LIN {X 0,Y 216.17,Z 835.857,A -85,B 0,C 180,E1 9801.223,E2 9801.223} C_VEL
LIN {X 0,Y 213.563,Z 840.911,A -85,B 0,C 180,E1 9796.189,E2 9796.189} C_VEL
LIN {X 0,Y 211.955,Z 844.646,A -85,B 0,C 180,E1 9790.637,E2 9790.637} C_VEL
LIN {X 0,Y 211.434,Z 846.63,A -85,B 0,C 180,E1 9785.221,E2 9785.221} C_VEL
LIN {X 0,Y 211.788,Z 847.099,A -85,B 0,C 180,E1 9779.975,E2 9779.975} C_VEL
LIN {X 0,Y 213.212,Z 845.891,A -85,B 0,C 180,E1 9774.219,E2 9774.219} C_VEL
LIN {X 0,Y 215.988,Z 842.864,A -85,B 0,C 180,E1 9768.553,E2 9768.553} C_VEL
LIN {X 0,Y 219.977,Z 838.26,A -85,B 0,C 180,E1 9763.339,E2 9763.339} C_VEL
LIN {X 0,Y 225.319,Z 832.008,A -85,B 0,C 180,E1 9758.406,E2 9758.406} C_VEL
LIN {X 0,Y 231.998,Z 823.945,A -85,B 0,C 180,E1 9753.723,E2 9753.723} C_VEL
LIN {X 0,Y 239.833,Z 814.067,A -85,B 0,C 180,E1 9749.394,E2 9749.394} C_VEL
LIN {X 0,Y 248.295,Z 802.757,A -85,B 0,C 180,E1 9745.582,E2 9745.582} C_VEL
LIN {X 0,Y 257.088,Z 790.107,A -85,B 0,C 180,E1 9742.245,E2 9742.245} C_VEL
LIN {X 0,Y 266.114,Z 775.981,A -85,B 0,C 180,E1 9739.307,E2 9739.307} C_VEL
LIN {X 0,Y 275.138,Z 760.195,A -85,B 0,C 180,E1 9736.725,E2 9736.725} C_VEL
LIN {X 0,Y 283.583,Z 743.647,A -85,B 0,C 180,E1 9734.582,E2 9734.582} C_VEL
LIN {X 0,Y 291.207,Z 726.587,A -85,B 0,C 180,E1 9732.821,E2 9732.821} C_VEL
LIN {X 0,Y 298.253,Z 708.268,A -85,B 0,C 180,E1 9731.326,E2 9731.326} C_VEL
LIN {X 0,Y 304.418,Z 689.211,A -85,B 0,C 180,E1 9730.108,E2 9730.108} C_VEL
LIN {X 0,Y 309.578,Z 669.056,A -85,B 0,C 180,E1 9729.137,E2 9729.137} C_VEL
LIN {X 0,Y 313.491,Z 648.587,A -85,B 0,C 180,E1 9728.428,E2 9728.428} C_VEL
LIN {X 0,Y 315.036,Z 637.769,A -85,B 0,C 180,E1 9728.146,E2 9728.146} C_VEL
LIN {X 0,Y 315.658,Z 630.27,A -85,B 0,C 180,E1 9727.794,E2 9727.794} C_VEL
LIN {X 0,Y 316.044,Z 610.74,A -85,B 0,C 180,E1 9726.277,E2 9726.277} C_VEL
LIN {X 0,Y 316.562,Z 604.27,A -85,B 0,C 180,E1 9726.008,E2 9726.008} C_VEL
LIN {X 0,Y 330.668,Z 479.091,A -85,B 0,C 180,E1 9723.364,E2 9723.364} C_VEL
LIN {X 0,Y 333.385,Z 441.647,A -85,B 0,C 180,E1 9721.202,E2 9721.202} C_VEL
LIN {X 0,Y 332.154,Z 436.517,A -85,B 0,C 180,E1 9718.878,E2 9718.878} C_VEL
LIN {X 0,Y 331.429,Z 432.32,A -85,B 0,C 180,E1 9716.107,E2 9716.107} C_VEL
LIN {X 0,Y 331.783,Z 429.625,A -85,B 0,C 180,E1 9712.38,E2 9712.38} C_VEL
LIN {X 0,Y 332.681,Z 430.118,A -85,B 0,C 180,E1 9710.135,E2 9710.135} C_VEL
LIN {X 0,Y 334.995,Z 433.817,A -85,B 0,C 180,E1 9706.801,E2 9706.801} C_VEL
LIN {X 0,Y 336.697,Z 436.983,A -85,B 0,C 180,E1 9705.066,E2 9705.066} C_VEL
LIN {X 0,Y 321.679,Z 592.371,A -85,B 0,C 180,E1 9701.883,E2 9701.883} C_VEL
LIN {X 0,Y 316.022,Z 652.978,A -85,B 0,C 180,E1 9700.612,E2 9700.612} C_VEL
LIN {X 0,Y 312.317,Z 675.121,A -85,B 0,C 180,E1 9699.999,E2 9699.999} C_VEL
LIN {X 0,Y 307.316,Z 696.218,A -85,B 0,C 180,E1 9699.228,E2 9699.228} C_VEL
LIN {X 0,Y 301.4,Z 716.25,A -85,B 0,C 180,E1 9698.252,E2 9698.252} C_VEL
LIN {X 0,Y 294.376,Z 735.972,A -85,B 0,C 180,E1 9697.008,E2 9697.008} C_VEL
LIN {X 0,Y 286.184,Z 755.614,A -85,B 0,C 180,E1 9695.432,E2 9695.432} C_VEL
LIN {X 0,Y 277.441,Z 774.165,A -85,B 0,C 180,E1 9693.569,E2 9693.569} C_VEL
LIN {X 0,Y 268.335,Z 791.382,A -85,B 0,C 180,E1 9691.402,E2 9691.402} C_VEL
LIN {X 0,Y 257.843,Z 809.537,A -85,B 0,C 180,E1 9688.546,E2 9688.546} C_VEL
LIN {X 0,Y 247.851,Z 825.668,A -85,B 0,C 180,E1 9685.377,E2 9685.377} C_VEL
LIN {X 0,Y 237.561,Z 841.407,A -85,B 0,C 180,E1 9681.47,E2 9681.47} C_VEL
LIN {X 0,Y 228.085,Z 855.483,A -85,B 0,C 180,E1 9677.057,E2 9677.057} C_VEL
LIN {X 0,Y 219.562,Z 868.331,A -85,B 0,C 180,E1 9672.018,E2 9672.018} C_VEL
LIN {X 0,Y 212.413,Z 879.754,A -85,B 0,C 180,E1 9666.373,E2 9666.373} C_VEL
LIN {X 0,Y 207.135,Z 889.148,A -85,B 0,C 180,E1 9660.45,E2 9660.45} C_VEL
LIN {X 0,Y 203.464,Z 897.482,A -85,B 0,C 180,E1 9653.76,E2 9653.76} C_VEL
LIN {X 0,Y 201.898,Z 903.094,A -85,B 0,C 180,E1 9647.878,E2 9647.878} C_VEL
LIN {X 0,Y 201.535,Z 907.332,A -85,B 0,C 180,E1 9641.733,E2 9641.733} C_VEL
LIN {X 0,Y 201.829,Z 909.538,A -85,B 0,C 180,E1 9636.825,E2 9636.825} C_VEL
LIN {X 0,Y 202.15,Z 910.582,A -85,B 0,C 180,E1 9632.265,E2 9632.265} C_VEL
LIN {X 0,Y 202.167,Z 910.586,A -85,B 0,C 180,E1 9628.013,E2 9628.013} C_VEL
LIN {X 0,Y 201.84,Z 909.458,A -85,B 0,C 180,E1 9623.169,E2 9623.169} C_VEL
LIN {X 0,Y 201.572,Z 906.678,A -85,B 0,C 180,E1 9617.682,E2 9617.682} C_VEL
LIN {X 0,Y 201.959,Z 902.561,A -85,B 0,C 180,E1 9612.122,E2 9612.122} C_VEL
LIN {X 0,Y 203.657,Z 896.224,A -85,B 0,C 180,E1 9605.948,E2 9605.948} C_VEL
LIN {X 0,Y 206.793,Z 888.559,A -85,B 0,C 180,E1 9600.128,E2 9600.128} C_VEL
LIN {X 0,Y 211.703,Z 878.744,A -85,B 0,C 180,E1 9594.326,E2 9594.326} C_VEL
LIN {X 0,Y 218.021,Z 867.475,A -85,B 0,C 180,E1 9589.016,E2 9589.016} C_VEL
LIN {X 0,Y 225.224,Z 855.274,A -85,B 0,C 180,E1 9584.375,E2 9584.375} C_VEL
LIN {X 0,Y 233.702,Z 840.845,A -85,B 0,C 180,E1 9580.016,E2 9580.016} C_VEL
LIN {X 0,Y 242.489,Z 825.468,A -85,B 0,C 180,E1 9576.279,E2 9576.279} C_VEL
LIN {X 0,Y 251.282,Z 809.376,A -85,B 0,C 180,E1 9573.117,E2 9573.117} C_VEL
LIN {X 0,Y 260.122,Z 791.762,A -85,B 0,C 180,E1 9570.349,E2 9570.349} C_VEL
LIN {X 0,Y 268.829,Z 772.701,A -85,B 0,C 180,E1 9567.946,E2 9567.946} C_VEL
LIN {X 0,Y 276.623,Z 753.661,A -85,B 0,C 180,E1 9566.014,E2 9566.014} C_VEL
LIN {X 0,Y 283.429,Z 734.543,A -85,B 0,C 180,E1 9564.47,E2 9564.47} C_VEL
LIN {X 0,Y 289.725,Z 713.651,A -85,B 0,C 180,E1 9563.138,E2 9563.138} C_VEL
LIN {X 0,Y 295.057,Z 692.142,A -85,B 0,C 180,E1 9562.083,E2 9562.083} C_VEL
LIN {X 0,Y 299.172,Z 670.359,A -85,B 0,C 180,E1 9561.305,E2 9561.305} C_VEL
LIN {X 0,Y 301.898,Z 648.014,A -85,B 0,C 180,E1 9560.706,E2 9560.706} C_VEL
LIN {X 0,Y 316.697,Z 449.988,A -85,B 0,C 180,E1 9556.577,E2 9556.577} C_VEL
LIN {X 0,Y 318.4,Z 427.647,A -85,B 0,C 180,E1 9556.089,E2 9556.089} C_VEL
LIN {X 0,Y 309.751,Z 414.232,A -85,B 0,C 180,E1 9552.443,E2 9552.443} C_VEL
LIN {X 0,Y 301.912,Z 402.88,A -85,B 0,C 180,E1 9548.667,E2 9548.667} C_VEL
LIN {X 0,Y 294.659,Z 393.174,A -85,B 0,C 180,E1 9544.574,E2 9544.574} C_VEL
LIN {X 0,Y 289.984,Z 387.27,A -85,B 0,C 180,E1 9541.492,E2 9541.492} C_VEL
LIN {X 0,Y 287.159,Z 383.801,A -85,B 0,C 180,E1 9539.402,E2 9539.402} C_VEL
LIN {X 0,Y 283.546,Z 379.395,A -85,B 0,C 180,E1 9536.337,E2 9536.337} C_VEL
LIN {X 0,Y 279.243,Z 374.32,A -85,B 0,C 180,E1 9531.766,E2 9531.766} C_VEL
LIN {X 0,Y 274.47,Z 369.423,A -85,B 0,C 180,E1 9523.057,E2 9523.057} C_VEL
LIN {X 0,Y 273.587,Z 369.085,A -85,B 0,C 180,E1 9519.238,E2 9519.238} C_VEL
LIN {X 0,Y 273.555,Z 370.592,A -85,B 0,C 180,E1 9514.915,E2 9514.915} C_VEL
LIN {X 0,Y 275.286,Z 373.534,A -85,B 0,C 180,E1 9509.075,E2 9509.075} C_VEL
LIN {X 0,Y 278.207,Z 378.589,A -85,B 0,C 180,E1 9504.141,E2 9504.141} C_VEL
LIN {X 0,Y 281.069,Z 383.491,A -85,B 0,C 180,E1 9500.642,E2 9500.642} C_VEL
LIN {X 0,Y 284.697,Z 389.345,A -85,B 0,C 180,E1 9497.191,E2 9497.191} C_VEL
LIN {X 0,Y 290.304,Z 398.667,A -85,B 0,C 180,E1 9492.892,E2 9492.892} C_VEL
LIN {X 0,Y 296.513,Z 409.789,A -85,B 0,C 180,E1 9488.915,E2 9488.915} C_VEL
LIN {X 0,Y 301.972,Z 420.129,A -85,B 0,C 180,E1 9485.903,E2 9485.903} C_VEL
LIN {X 0,Y 303.039,Z 422.43,A -85,B 0,C 180,E1 9485.339,E2 9485.339} C_VEL
LIN {X 0,Y 302.745,Z 475.251,A -85,B 0,C 180,E1 9482.474,E2 9482.474} C_VEL
LIN {X 0,Y 287.453,Z 637.405,A -85,B 0,C 180,E1 9478.809,E2 9478.809} C_VEL
LIN {X 0,Y 284.269,Z 658.885,A -85,B 0,C 180,E1 9478.1,E2 9478.1} C_VEL
LIN {X 0,Y 280.102,Z 679.277,A -85,B 0,C 180,E1 9477.133,E2 9477.133} C_VEL
LIN {X 0,Y 274.985,Z 699.045,A -85,B 0,C 180,E1 9475.872,E2 9475.872} C_VEL
LIN {X 0,Y 268.872,Z 718.482,A -85,B 0,C 180,E1 9474.265,E2 9474.265} C_VEL
LIN {X 0,Y 262.041,Z 736.952,A -85,B 0,C 180,E1 9472.315,E2 9472.315} C_VEL
LIN {X 0,Y 255.013,Z 753.63,A -85,B 0,C 180,E1 9470.102,E2 9470.102} C_VEL
LIN {X 0,Y 247.357,Z 769.856,A -85,B 0,C 180,E1 9467.407,E2 9467.407} C_VEL
LIN {X 0,Y 239.545,Z 784.904,A -85,B 0,C 180,E1 9464.259,E2 9464.259} C_VEL
LIN {X 0,Y 231.944,Z 798.441,A -85,B 0,C 180,E1 9460.685,E2 9460.685} C_VEL
LIN {X 0,Y 224.761,Z 810.489,A -85,B 0,C 180,E1 9456.644,E2 9456.644} C_VEL
LIN {X 0,Y 218.603,Z 820.494,A -85,B 0,C 180,E1 9452.362,E2 9452.362} C_VEL
LIN {X 0,Y 213.219,Z 829.191,A -85,B 0,C 180,E1 9447.584,E2 9447.584} C_VEL
LIN {X 0,Y 208.872,Z 836.46,A -85,B 0,C 180,E1 9442.3,E2 9442.3} C_VEL
LIN {X 0,Y 205.878,Z 841.925,A -85,B 0,C 180,E1 9436.809,E2 9436.809} C_VEL
LIN {X 0,Y 204.138,Z 845.701,A -85,B 0,C 180,E1 9431.143,E2 9431.143} C_VEL
LIN {X 0,Y 203.54,Z 847.784,A -85,B 0,C 180,E1 9425.633,E2 9425.633} C_VEL
LIN {X 0,Y 203.88,Z 848.366,A -85,B 0,C 180,E1 9419.989,E2 9419.989} C_VEL
LIN {X 0,Y 205.28,Z 847.317,A -85,B 0,C 180,E1 9414.237,E2 9414.237} C_VEL
LIN {X 0,Y 207.877,Z 844.743,A -85,B 0,C 180,E1 9408.784,E2 9408.784} C_VEL
LIN {X 0,Y 212.139,Z 840.256,A -85,B 0,C 180,E1 9403.109,E2 9403.109} C_VEL
LIN {X 0,Y 217.821,Z 834.105,A -85,B 0,C 180,E1 9397.864,E2 9397.864} C_VEL
LIN {X 0,Y 224.554,Z 826.561,A -85,B 0,C 180,E1 9393.171,E2 9393.171} C_VEL
LIN {X 0,Y 232.615,Z 817.088,A -85,B 0,C 180,E1 9388.74,E2 9388.74} C_VEL
LIN {X 0,Y 241.689,Z 805.725,A -85,B 0,C 180,E1 9384.697,E2 9384.697} C_VEL
LIN {X 0,Y 251.331,Z 792.624,A -85,B 0,C 180,E1 9381.117,E2 9381.117} C_VEL
LIN {X 0,Y 261.187,Z 777.895,A -85,B 0,C 180,E1 9378.001,E2 9378.001} C_VEL
LIN {X 0,Y 270.309,Z 762.74,A -85,B 0,C 180,E1 9375.483,E2 9375.483} C_VEL
LIN {X 0,Y 278.993,Z 746.565,A -85,B 0,C 180,E1 9373.355,E2 9373.355} C_VEL
LIN {X 0,Y 287.238,Z 729.113,A -85,B 0,C 180,E1 9371.525,E2 9371.525} C_VEL
LIN {X 0,Y 294.72,Z 710.666,A -85,B 0,C 180,E1 9370.005,E2 9370.005} C_VEL
LIN {X 0,Y 301.126,Z 691.612,A -85,B 0,C 180,E1 9368.785,E2 9368.785} C_VEL
LIN {X 0,Y 306.508,Z 671.619,A -85,B 0,C 180,E1 9367.814,E2 9367.814} C_VEL
LIN {X 0,Y 310.78,Z 650.649,A -85,B 0,C 180,E1 9367.078,E2 9367.078} C_VEL
LIN {X 0,Y 314.401,Z 623.419,A -85,B 0,C 180,E1 9366.425,E2 9366.425} C_VEL
LIN {X 0,Y 316.562,Z 604.27,A -85,B 0,C 180,E1 9366.008,E2 9366.008} C_VEL
LIN {X 0,Y 317.157,Z 596.754,A -85,B 0,C 180,E1 9365.672,E2 9365.672} C_VEL
LIN {X 0,Y 317.86,Z 577.246,A -85,B 0,C 180,E1 9364.157,E2 9364.157} C_VEL
LIN {X 0,Y 318.435,Z 570.779,A -85,B 0,C 180,E1 9363.89,E2 9363.89} C_VEL
LIN {X 0,Y 328.867,Z 480.612,A -85,B 0,C 180,E1 9362.03,E2 9362.03} C_VEL
LIN {X 0,Y 331.591,Z 447.558,A -85,B 0,C 180,E1 9360.129,E2 9360.129} C_VEL
LIN {X 0,Y 330.72,Z 443.262,A -85,B 0,C 180,E1 9358.007,E2 9358.007} C_VEL
LIN {X 0,Y 330.277,Z 439.803,A -85,B 0,C 180,E1 9355.485,E2 9355.485} C_VEL
LIN {X 0,Y 330.749,Z 437.558,A -85,B 0,C 180,E1 9352.356,E2 9352.356} C_VEL
LIN {X 0,Y 331.567,Z 438.023,A -85,B 0,C 180,E1 9350.277,E2 9350.277} C_VEL
LIN {X 0,Y 333.735,Z 441.661,A -85,B 0,C 180,E1 9347.014,E2 9347.014} C_VEL
LIN {X 0,Y 334.381,Z 443.09,A -85,B 0,C 180,E1 9346.283,E2 9346.283} C_VEL
LIN {X 0,Y 318.47,Z 601.078,A -85,B 0,C 180,E1 9343.076,E2 9343.076} C_VEL
LIN {X 0,Y 313.439,Z 652.552,A -85,B 0,C 180,E1 9342.001,E2 9342.001} C_VEL
LIN {X 0,Y 309.591,Z 674.771,A -85,B 0,C 180,E1 9341.396,E2 9341.396} C_VEL
LIN {X 0,Y 304.391,Z 696.001,A -85,B 0,C 180,E1 9340.635,E2 9340.635} C_VEL
LIN {X 0,Y 297.952,Z 717.011,A -85,B 0,C 180,E1 9339.624,E2 9339.624} C_VEL
LIN {X 0,Y 290.796,Z 736.37,A -85,B 0,C 180,E1 9338.413,E2 9338.413} C_VEL
LIN {X 0,Y 282.261,Z 755.989,A -85,B 0,C 180,E1 9336.846,E2 9336.846} C_VEL
LIN {X 0,Y 272.72,Z 775.311,A -85,B 0,C 180,E1 9334.893,E2 9334.893} C_VEL
LIN {X 0,Y 262.541,Z 793.752,A -85,B 0,C 180,E1 9332.536,E2 9332.536} C_VEL
LIN {X 0,Y 252.197,Z 810.653,A -85,B 0,C 180,E1 9329.795,E2 9329.795} C_VEL
LIN {X 0,Y 241.257,Z 827.303,A -85,B 0,C 180,E1 9326.404,E2 9326.404} C_VEL
LIN {X 0,Y 231.29,Z 841.831,A -85,B 0,C 180,E1 9322.69,E2 9322.69} C_VEL
LIN {X 0,Y 221.37,Z 855.737,A -85,B 0,C 180,E1 9318.176,E2 9318.176} C_VEL
LIN {X 0,Y 212.468,Z 868.298,A -85,B 0,C 180,E1 9313.024,E2 9313.024} C_VEL
LIN {X 0,Y 205.199,Z 879.188,A -85,B 0,C 180,E1 9307.416,E2 9307.416} C_VEL
LIN {X 0,Y 199.432,Z 888.758,A -85,B 0,C 180,E1 9301.087,E2 9301.087} C_VEL
LIN {X 0,Y 195.696,Z 896.562,A -85,B 0,C 180,E1 9294.443,E2 9294.443} C_VEL
LIN {X 0,Y 193.939,Z 902.385,A -85,B 0,C 180,E1 9288.016,E2 9288.016} C_VEL
LIN {X 0,Y 193.589,Z 906.259,A -85,B 0,C 180,E1 9281.92,E2 9281.92} C_VEL
LIN {X 0,Y 193.903,Z 908.416,A -85,B 0,C 180,E1 9276.808,E2 9276.808} C_VEL
LIN {X 0,Y 194.248,Z 909.402,A -85,B 0,C 180,E1 9272.062,E2 9272.062} C_VEL
LIN {X 0,Y 194.242,Z 909.331,A -85,B 0,C 180,E1 9267.637,E2 9267.637} C_VEL
LIN {X 0,Y 193.896,Z 908.166,A -85,B 0,C 180,E1 9262.888,E2 9262.888} C_VEL
LIN {X 0,Y 193.633,Z 905.493,A -85,B 0,C 180,E1 9257.407,E2 9257.407} C_VEL
LIN {X 0,Y 194.065,Z 901.416,A -85,B 0,C 180,E1 9251.68,E2 9251.68} C_VEL
LIN {X 0,Y 195.909,Z 895.08,A -85,B 0,C 180,E1 9245.257,E2 9245.257} C_VEL
LIN {X 0,Y 199.429,Z 887.119,A -85,B 0,C 180,E1 9239.019,E2 9239.019} C_VEL
LIN {X 0,Y 204.4,Z 877.821,A -85,B 0,C 180,E1 9233.345,E2 9233.345} C_VEL
LIN {X 0,Y 211.227,Z 866.278,A -85,B 0,C 180,E1 9227.762,E2 9227.762} C_VEL
LIN {X 0,Y 219.205,Z 853.421,A -85,B 0,C 180,E1 9222.816,E2 9222.816} C_VEL
LIN {X 0,Y 227.817,Z 839.442,A -85,B 0,C 180,E1 9218.552,E2 9218.552} C_VEL
LIN {X 0,Y 236.868,Z 824.136,A -85,B 0,C 180,E1 9214.826,E2 9214.826} C_VEL
LIN {X 0,Y 246.172,Z 807.637,A -85,B 0,C 180,E1 9211.598,E2 9211.598} C_VEL
LIN {X 0,Y 255.095,Z 790.434,A -85,B 0,C 180,E1 9208.902,E2 9208.902} C_VEL
LIN {X 0,Y 263.573,Z 772.389,A -85,B 0,C 180,E1 9206.633,E2 9206.633} C_VEL
LIN {X 0,Y 271.763,Z 752.873,A -85,B 0,C 180,E1 9204.663,E2 9204.663} C_VEL
LIN {X 0,Y 278.843,Z 733.4,A -85,B 0,C 180,E1 9203.108,E2 9203.108} C_VEL
LIN {X 0,Y 285.119,Z 712.991,A -85,B 0,C 180,E1 9201.822,E2 9201.822} C_VEL
LIN {X 0,Y 290.521,Z 691.722,A -85,B 0,C 180,E1 9200.788,E2 9200.788} C_VEL
LIN {X 0,Y 294.733,Z 669.928,A -85,B 0,C 180,E1 9200.015,E2 9200.015} C_VEL
LIN {X 0,Y 297.515,Z 647.659,A -85,B 0,C 180,E1 9199.42,E2 9199.42} C_VEL
LIN {X 0,Y 313.189,Z 444.677,A -85,B 0,C 180,E1 9195.196,E2 9195.196} C_VEL
LIN {X 0,Y 314.111,Z 432.001,A -85,B 0,C 180,E1 9194.895,E2 9194.895} C_VEL
LIN {X 0,Y 305.768,Z 418.915,A -85,B 0,C 180,E1 9191.181,E2 9191.181} C_VEL
LIN {X 0,Y 298.708,Z 408.748,A -85,B 0,C 180,E1 9187.598,E2 9187.598} C_VEL
LIN {X 0,Y 292.303,Z 400.006,A -85,B 0,C 180,E1 9183.825,E2 9183.825} C_VEL
LIN {X 0,Y 287.642,Z 393.945,A -85,B 0,C 180,E1 9180.598,E2 9180.598} C_VEL
LIN {X 0,Y 282.377,Z 387.342,A -85,B 0,C 180,E1 9176.245,E2 9176.245} C_VEL
LIN {X 0,Y 277.985,Z 382.142,A -85,B 0,C 180,E1 9171.521,E2 9171.521} C_VEL
LIN {X 0,Y 273.397,Z 377.349,A -85,B 0,C 180,E1 9162.989,E2 9162.989} C_VEL
LIN {X 0,Y 272.532,Z 377.032,A -85,B 0,C 180,E1 9159.154,E2 9159.154} C_VEL
LIN {X 0,Y 272.507,Z 378.603,A -85,B 0,C 180,E1 9154.811,E2 9154.811} C_VEL
LIN {X 0,Y 274.071,Z 381.257,A -85,B 0,C 180,E1 9149.429,E2 9149.429} C_VEL
LIN {X 0,Y 276.883,Z 386.353,A -85,B 0,C 180,E1 9144.453,E2 9144.453} C_VEL
LIN {X 0,Y 279.604,Z 391.183,A -85,B 0,C 180,E1 9140.998,E2 9140.998} C_VEL
LIN {X 0,Y 283.619,Z 397.734,A -85,B 0,C 180,E1 9137.127,E2 9137.127} C_VEL
LIN {X 0,Y 289.363,Z 407.859,A -85,B 0,C 180,E1 9132.683,E2 9132.683} C_VEL
LIN {X 0,Y 295.031,Z 418.35,A -85,B 0,C 180,E1 9129.022,E2 9129.022} C_VEL
LIN {X 0,Y 299.492,Z 427.256,A -85,B 0,C 180,E1 9126.491,E2 9126.491} C_VEL
LIN {X 0,Y 298.901,Z 476.534,A -85,B 0,C 180,E1 9123.797,E2 9123.797} C_VEL
LIN {X 0,Y 283.243,Z 638.046,A -85,B 0,C 180,E1 9120.17,E2 9120.17} C_VEL
LIN {X 0,Y 279.986,Z 659.378,A -85,B 0,C 180,E1 9119.469,E2 9119.469} C_VEL
LIN {X 0,Y 275.637,Z 680.044,A -85,B 0,C 180,E1 9118.492,E2 9118.492} C_VEL
LIN {X 0,Y 270.204,Z 700.343,A -85,B 0,C 180,E1 9117.196,E2 9117.196} C_VEL
LIN {X 0,Y 263.615,Z 720.487,A -85,B 0,C 180,E1 9115.513,E2 9115.513} C_VEL
LIN {X 0,Y 256.549,Z 738.817,A -85,B 0,C 180,E1 9113.548,E2 9113.548} C_VEL
LIN {X 0,Y 248.663,Z 756.656,A -85,B 0,C 180,E1 9111.119,E2 9111.119} C_VEL
LIN {X 0,Y 240.539,Z 773.015,A -85,B 0,C 180,E1 9108.293,E2 9108.293} C_VEL
LIN {X 0,Y 232.765,Z 787.271,A -85,B 0,C 180,E1 9105.193,E2 9105.193} C_VEL
LIN {X 0,Y 224.916,Z 800.605,A -85,B 0,C 180,E1 9101.542,E2 9101.542} C_VEL
LIN {X 0,Y 217.496,Z 812.502,A -85,B 0,C 180,E1 9097.398,E2 9097.398} C_VEL
LIN {X 0,Y 210.783,Z 822.92,A -85,B 0,C 180,E1 9092.722,E2 9092.722} C_VEL
LIN {X 0,Y 205.001,Z 831.807,A -85,B 0,C 180,E1 9087.487,E2 9087.487} C_VEL
LIN {X 0,Y 200.655,Z 838.738,A -85,B 0,C 180,E1 9081.983,E2 9081.983} C_VEL
LIN {X 0,Y 197.824,Z 843.652,A -85,B 0,C 180,E1 9076.559,E2 9076.559} C_VEL
LIN {X 0,Y 196.185,Z 847.084,A -85,B 0,C 180,E1 9070.967,E2 9070.967} C_VEL
LIN {X 0,Y 195.622,Z 849.078,A -85,B 0,C 180,E1 9065.225,E2 9065.225} C_VEL
LIN {X 0,Y 196.072,Z 849.607,A -85,B 0,C 180,E1 9059.344,E2 9059.344} C_VEL
LIN {X 0,Y 197.684,Z 848.507,A -85,B 0,C 180,E1 9053.361,E2 9053.361} C_VEL
LIN {X 0,Y 200.79,Z 845.675,A -85,B 0,C 180,E1 9047.377,E2 9047.377} C_VEL
LIN {X 0,Y 205.271,Z 841.288,A -85,B 0,C 180,E1 9041.825,E2 9041.825} C_VEL
LIN {X 0,Y 211.383,Z 835.125,A -85,B 0,C 180,E1 9036.481,E2 9036.481} C_VEL
LIN {X 0,Y 218.576,Z 827.548,A -85,B 0,C 180,E1 9031.703,E2 9031.703} C_VEL
LIN {X 0,Y 227.116,Z 818.079,A -85,B 0,C 180,E1 9027.223,E2 9027.223} C_VEL
LIN {X 0,Y 236.255,Z 807.245,A -85,B 0,C 180,E1 9023.319,E2 9023.319} C_VEL
LIN {X 0,Y 246.454,Z 794.059,A -85,B 0,C 180,E1 9019.677,E2 9019.677} C_VEL
LIN {X 0,Y 256.252,Z 780.104,A -85,B 0,C 180,E1 9016.694,E2 9016.694} C_VEL
LIN {X 0,Y 265.975,Z 764.732,A -85,B 0,C 180,E1 9014.111,E2 9014.111} C_VEL
LIN {X 0,Y 275.374,Z 748.031,A -85,B 0,C 180,E1 9011.908,E2 9011.908} C_VEL
LIN {X 0,Y 283.81,Z 730.858,A -85,B 0,C 180,E1 9010.117,E2 9010.117} C_VEL
LIN {X 0,Y 291.715,Z 712.171,A -85,B 0,C 180,E1 9008.586,E2 9008.586} C_VEL
LIN {X 0,Y 298.41,Z 692.969,A -85,B 0,C 180,E1 9007.37,E2 9007.37} C_VEL
LIN {X 0,Y 303.96,Z 673.133,A -85,B 0,C 180,E1 9006.417,E2 9006.417} C_VEL
LIN {X 0,Y 308.455,Z 651.86,A -85,B 0,C 180,E1 9005.677,E2 9005.677} C_VEL
LIN {X 0,Y 311.884,Z 627.446,A -85,B 0,C 180,E1 9005.092,E2 9005.092} C_VEL
LIN {X 0,Y 318.435,Z 570.779,A -85,B 0,C 180,E1 9003.89,E2 9003.89} C_VEL
LIN {X 0,Y 319.094,Z 563.262,A -85,B 0,C 180,E1 9003.56,E2 9003.56} C_VEL
LIN {X 0,Y 320.151,Z 543.752,A -85,B 0,C 180,E1 9002.062,E2 9002.062} C_VEL
LIN {X 0,Y 320.783,Z 537.287,A -85,B 0,C 180,E1 9001.799,E2 9001.799} C_VEL
LIN {X 0,Y 327.345,Z 482.115,A -85,B 0,C 180,E1 9000.678,E2 9000.678} C_VEL
LIN {X 0,Y 329.964,Z 453.53,A -85,B 0,C 180,E1 8999.044,E2 8999.044} C_VEL
LIN {X 0,Y 329.304,Z 449.178,A -85,B 0,C 180,E1 8996.518,E2 8996.518} C_VEL
LIN {X 0,Y 329.219,Z 447.394,A -85,B 0,C 180,E1 8994.947,E2 8994.947} C_VEL
LIN {X 0,Y 329.764,Z 445.497,A -85,B 0,C 180,E1 8992.157,E2 8992.157} C_VEL
LIN {X 0,Y 330.455,Z 445.928,A -85,B 0,C 180,E1 8990.42,E2 8990.42} C_VEL
LIN {X 0,Y 332.259,Z 449.007,A -85,B 0,C 180,E1 8987.525,E2 8987.525} C_VEL
LIN {X 0,Y 316.052,Z 604.122,A -85,B 0,C 180,E1 8984.412,E2 8984.412} C_VEL
LIN {X 0,Y 311.048,Z 652.363,A -85,B 0,C 180,E1 8983.41,E2 8983.41} C_VEL
LIN {X 0,Y 306.925,Z 675.367,A -85,B 0,C 180,E1 8982.794,E2 8982.794} C_VEL
LIN {X 0,Y 301.615,Z 696.234,A -85,B 0,C 180,E1 8982.057,E2 8982.057} C_VEL
LIN {X 0,Y 294.911,Z 717.227,A -85,B 0,C 180,E1 8981.061,E2 8981.061} C_VEL
LIN {X 0,Y 287.146,Z 737.471,A -85,B 0,C 180,E1 8979.808,E2 8979.808} C_VEL
LIN {X 0,Y 278.558,Z 756.406,A -85,B 0,C 180,E1 8978.302,E2 8978.302} C_VEL
LIN {X 0,Y 268.525,Z 775.823,A -85,B 0,C 180,E1 8976.339,E2 8976.339} C_VEL
LIN {X 0,Y 258.219,Z 793.739,A -85,B 0,C 180,E1 8974.052,E2 8974.052} C_VEL
LIN {X 0,Y 247.366,Z 810.743,A -85,B 0,C 180,E1 8971.29,E2 8971.29} C_VEL
LIN {X 0,Y 236.673,Z 826.276,A -85,B 0,C 180,E1 8968.114,E2 8968.114} C_VEL
LIN {X 0,Y 225.636,Z 841.512,A -85,B 0,C 180,E1 8964.181,E2 8964.181} C_VEL
LIN {X 0,Y 215.253,Z 855.308,A -85,B 0,C 180,E1 8959.617,E2 8959.617} C_VEL
LIN {X 0,Y 205.868,Z 867.72,A -85,B 0,C 180,E1 8954.373,E2 8954.373} C_VEL
LIN {X 0,Y 197.92,Z 878.789,A -85,B 0,C 180,E1 8948.412,E2 8948.412} C_VEL
LIN {X 0,Y 191.989,Z 887.968,A -85,B 0,C 180,E1 8942.083,E2 8942.083} C_VEL
LIN {X 0,Y 187.953,Z 895.653,A -85,B 0,C 180,E1 8935.183,E2 8935.183} C_VEL
LIN {X 0,Y 186.037,Z 901.378,A -85,B 0,C 180,E1 8928.484,E2 8928.484} C_VEL
LIN {X 0,Y 185.64,Z 905.189,A -85,B 0,C 180,E1 8922.122,E2 8922.122} C_VEL
LIN {X 0,Y 186.005,Z 907.397,A -85,B 0,C 180,E1 8916.478,E2 8916.478} C_VEL
LIN {X 0,Y 186.356,Z 908.255,A -85,B 0,C 180,E1 8911.534,E2 8911.534} C_VEL
LIN {X 0,Y 186.297,Z 907.992,A -85,B 0,C 180,E1 8906.92,E2 8906.92} C_VEL
LIN {X 0,Y 185.897,Z 906.609,A -85,B 0,C 180,E1 8901.958,E2 8901.958} C_VEL
LIN {X 0,Y 185.704,Z 903.996,A -85,B 0,C 180,E1 8896.61,E2 8896.61} C_VEL
LIN {X 0,Y 186.359,Z 899.499,A -85,B 0,C 180,E1 8890.241,E2 8890.241} C_VEL
LIN {X 0,Y 188.474,Z 893.246,A -85,B 0,C 180,E1 8883.873,E2 8883.873} C_VEL
LIN {X 0,Y 192.574,Z 884.825,A -85,B 0,C 180,E1 8877.259,E2 8877.259} C_VEL
LIN {X 0,Y 198.262,Z 875.111,A -85,B 0,C 180,E1 8871.289,E2 8871.289} C_VEL
LIN {X 0,Y 205.361,Z 863.805,A -85,B 0,C 180,E1 8865.871,E2 8865.871} C_VEL
LIN {X 0,Y 214.031,Z 850.47,A -85,B 0,C 180,E1 8860.814,E2 8860.814} C_VEL
LIN {X 0,Y 223.017,Z 836.507,A -85,B 0,C 180,E1 8856.605,E2 8856.605} C_VEL
LIN {X 0,Y 232.625,Z 820.799,A -85,B 0,C 180,E1 8852.874,E2 8852.874} C_VEL
LIN {X 0,Y 242.348,Z 803.855,A -85,B 0,C 180,E1 8849.676,E2 8849.676} C_VEL
LIN {X 0,Y 251.5,Z 786.521,A -85,B 0,C 180,E1 8847.056,E2 8847.056} C_VEL
LIN {X 0,Y 260.092,Z 768.366,A -85,B 0,C 180,E1 8844.869,E2 8844.869} C_VEL
LIN {X 0,Y 268.282,Z 748.836,A -85,B 0,C 180,E1 8842.991,E2 8842.991} C_VEL
LIN {X 0,Y 275.581,Z 728.841,A -85,B 0,C 180,E1 8841.463,E2 8841.463} C_VEL
LIN {X 0,Y 281.672,Z 708.831,A -85,B 0,C 180,E1 8840.275,E2 8840.275} C_VEL
LIN {X 0,Y 287.058,Z 686.949,A -85,B 0,C 180,E1 8839.291,E2 8839.291} C_VEL
LIN {X 0,Y 291.123,Z 665.006,A -85,B 0,C 180,E1 8838.557,E2 8838.557} C_VEL
LIN {X 0,Y 293.641,Z 642.995,A -85,B 0,C 180,E1 8838.003,E2 8838.003} C_VEL
LIN {X 0,Y 308.705,Z 453.171,A -85,B 0,C 180,E1 8834.071,E2 8834.071} C_VEL
LIN {X 0,Y 310.051,Z 436.581,A -85,B 0,C 180,E1 8833.712,E2 8833.712} C_VEL
LIN {X 0,Y 302.588,Z 424.787,A -85,B 0,C 180,E1 8830.231,E2 8830.231} C_VEL
LIN {X 0,Y 295.607,Z 414.546,A -85,B 0,C 180,E1 8826.507,E2 8826.507} C_VEL
LIN {X 0,Y 289.855,Z 406.626,A -85,B 0,C 180,E1 8822.967,E2 8822.967} C_VEL
LIN {X 0,Y 284.558,Z 399.648,A -85,B 0,C 180,E1 8819.095,E2 8819.095} C_VEL
LIN {X 0,Y 280.532,Z 394.641,A -85,B 0,C 180,E1 8815.504,E2 8815.504} C_VEL
LIN {X 0,Y 276.563,Z 389.834,A -85,B 0,C 180,E1 8811.057,E2 8811.057} C_VEL
LIN {X 0,Y 272.262,Z 385.191,A -85,B 0,C 180,E1 8802.696,E2 8802.696} C_VEL
LIN {X 0,Y 271.45,Z 385.023,A -85,B 0,C 180,E1 8798.737,E2 8798.737} C_VEL
LIN {X 0,Y 272.265,Z 388.16,A -85,B 0,C 180,E1 8791.369,E2 8791.369} C_VEL
LIN {X 0,Y 272.958,Z 389.294,A -85,B 0,C 180,E1 8789.503,E2 8789.503} C_VEL
LIN {X 0,Y 275.484,Z 393.952,A -85,B 0,C 180,E1 8784.883,E2 8784.883} C_VEL
LIN {X 0,Y 278.105,Z 398.787,A -85,B 0,C 180,E1 8781.409,E2 8781.409} C_VEL
LIN {X 0,Y 281.96,Z 405.288,A -85,B 0,C 180,E1 8777.568,E2 8777.568} C_VEL
LIN {X 0,Y 287.366,Z 415.128,A -85,B 0,C 180,E1 8773.219,E2 8773.219} C_VEL
LIN {X 0,Y 292.962,Z 425.805,A -85,B 0,C 180,E1 8769.482,E2 8769.482} C_VEL
LIN {X 0,Y 296.022,Z 432.23,A -85,B 0,C 180,E1 8767.659,E2 8767.659} C_VEL
LIN {X 0,Y 295.207,Z 477.891,A -85,B 0,C 180,E1 8765.153,E2 8765.153} C_VEL
LIN {X 0,Y 279.222,Z 638.478,A -85,B 0,C 180,E1 8761.576,E2 8761.576} C_VEL
LIN {X 0,Y 275.866,Z 659.866,A -85,B 0,C 180,E1 8760.879,E2 8760.879} C_VEL
LIN {X 0,Y 271.332,Z 680.804,A -85,B 0,C 180,E1 8759.896,E2 8759.896} C_VEL
LIN {X 0,Y 265.916,Z 700.494,A -85,B 0,C 180,E1 8758.649,E2 8758.649} C_VEL
LIN {X 0,Y 259.206,Z 720.515,A -85,B 0,C 180,E1 8756.997,E2 8756.997} C_VEL
LIN {X 0,Y 251.825,Z 739.155,A -85,B 0,C 180,E1 8755.017,E2 8755.017} C_VEL
LIN {X 0,Y 243.912,Z 756.566,A -85,B 0,C 180,E1 8752.667,E2 8752.667} C_VEL
LIN {X 0,Y 235.807,Z 772.452,A -85,B 0,C 180,E1 8749.961,E2 8749.961} C_VEL
LIN {X 0,Y 227.666,Z 786.953,A -85,B 0,C 180,E1 8746.852,E2 8746.852} C_VEL
LIN {X 0,Y 219.407,Z 800.499,A -85,B 0,C 180,E1 8743.173,E2 8743.173} C_VEL
LIN {X 0,Y 211.542,Z 812.561,A -85,B 0,C 180,E1 8738.976,E2 8738.976} C_VEL
LIN {X 0,Y 204.373,Z 823.143,A -85,B 0,C 180,E1 8734.211,E2 8734.211} C_VEL
LIN {X 0,Y 198.441,Z 831.766,A -85,B 0,C 180,E1 8729.137,E2 8729.137} C_VEL
LIN {X 0,Y 193.836,Z 838.643,A -85,B 0,C 180,E1 8723.784,E2 8723.784} C_VEL
LIN {X 0,Y 190.345,Z 844.315,A -85,B 0,C 180,E1 8717.689,E2 8717.689} C_VEL
LIN {X 0,Y 188.429,Z 848.025,A -85,B 0,C 180,E1 8711.759,E2 8711.759} C_VEL
LIN {X 0,Y 187.731,Z 850.207,A -85,B 0,C 180,E1 8705.793,E2 8705.793} C_VEL
LIN {X 0,Y 188.155,Z 850.875,A -85,B 0,C 180,E1 8699.412,E2 8699.412} C_VEL
LIN {X 0,Y 189.813,Z 849.896,A -85,B 0,C 180,E1 8693.192,E2 8693.192} C_VEL
LIN {X 0,Y 192.887,Z 847.374,A -85,B 0,C 180,E1 8687.235,E2 8687.235} C_VEL
LIN {X 0,Y 197.822,Z 842.969,A -85,B 0,C 180,E1 8681.146,E2 8681.146} C_VEL
LIN {X 0,Y 204.237,Z 836.982,A -85,B 0,C 180,E1 8675.63,E2 8675.63} C_VEL
LIN {X 0,Y 211.929,Z 829.451,A -85,B 0,C 180,E1 8670.631,E2 8670.631} C_VEL
LIN {X 0,Y 220.909,Z 820.103,A -85,B 0,C 180,E1 8666.041,E2 8666.041} C_VEL
LIN {X 0,Y 231.059,Z 808.7,A -85,B 0,C 180,E1 8661.847,E2 8661.847} C_VEL
LIN {X 0,Y 241.216,Z 796.197,A -85,B 0,C 180,E1 8658.347,E2 8658.347} C_VEL
LIN {X 0,Y 251.422,Z 782.429,A -85,B 0,C 180,E1 8655.35,E2 8655.35} C_VEL
LIN {X 0,Y 261.846,Z 766.752,A -85,B 0,C 180,E1 8652.689,E2 8652.689} C_VEL
LIN {X 0,Y 271.512,Z 750.369,A -85,B 0,C 180,E1 8650.519,E2 8650.519} C_VEL
LIN {X 0,Y 280.212,Z 733.574,A -85,B 0,C 180,E1 8648.755,E2 8648.755} C_VEL
LIN {X 0,Y 288.524,Z 714.639,A -85,B 0,C 180,E1 8647.206,E2 8647.206} C_VEL
LIN {X 0,Y 295.557,Z 695.429,A -85,B 0,C 180,E1 8645.988,E2 8645.988} C_VEL
LIN {X 0,Y 301.594,Z 674.946,A -85,B 0,C 180,E1 8645.005,E2 8645.005} C_VEL
LIN {X 0,Y 306.247,Z 654.078,A -85,B 0,C 180,E1 8644.28,E2 8644.28} C_VEL
LIN {X 0,Y 309.558,Z 632.237,A -85,B 0,C 180,E1 8643.749,E2 8643.749} C_VEL
LIN {X 0,Y 320.783,Z 537.287,A -85,B 0,C 180,E1 8641.799,E2 8641.799} C_VEL
LIN {X 0,Y 321.519,Z 529.774,A -85,B 0,C 180,E1 8641.473,E2 8641.473} C_VEL
LIN {X 0,Y 322.92,Z 510.28,A -85,B 0,C 180,E1 8639.99,E2 8639.99} C_VEL
LIN {X 0,Y 323.606,Z 503.816,A -85,B 0,C 180,E1 8639.734,E2 8639.734} C_VEL
LIN {X 0,Y 326.065,Z 483.544,A -85,B 0,C 180,E1 8639.306,E2 8639.306} C_VEL
LIN {X 0,Y 328.48,Z 459.646,A -85,B 0,C 180,E1 8637.95,E2 8637.95} C_VEL
LIN {X 0,Y 328.148,Z 455.644,A -85,B 0,C 180,E1 8635.28,E2 8635.28} C_VEL
LIN {X 0,Y 328.731,Z 453.431,A -85,B 0,C 180,E1 8632.133,E2 8632.133} C_VEL
LIN {X 0,Y 329.346,Z 453.831,A -85,B 0,C 180,E1 8630.564,E2 8630.564} C_VEL
LIN {X 0,Y 330.275,Z 455.867,A -85,B 0,C 180,E1 8628.76,E2 8628.76} C_VEL
LIN {X 0,Y 313.519,Z 610.111,A -85,B 0,C 180,E1 8625.71,E2 8625.71} C_VEL
LIN {X 0,Y 308.858,Z 652.66,A -85,B 0,C 180,E1 8624.833,E2 8624.833} C_VEL
LIN {X 0,Y 304.72,Z 674.989,A -85,B 0,C 180,E1 8624.247,E2 8624.247} C_VEL
LIN {X 0,Y 299.226,Z 695.919,A -85,B 0,C 180,E1 8623.528,E2 8623.528} C_VEL
LIN {X 0,Y 292.373,Z 716.748,A -85,B 0,C 180,E1 8622.569,E2 8622.569} C_VEL
LIN {X 0,Y 284.799,Z 736.045,A -85,B 0,C 180,E1 8621.416,E2 8621.416} C_VEL
LIN {X 0,Y 276.034,Z 754.845,A -85,B 0,C 180,E1 8619.971,E2 8619.971} C_VEL
LIN {X 0,Y 265.69,Z 774.378,A -85,B 0,C 180,E1 8618.062,E2 8618.062} C_VEL
LIN {X 0,Y 255.248,Z 791.981,A -85,B 0,C 180,E1 8615.875,E2 8615.875} C_VEL
LIN {X 0,Y 243.785,Z 809.306,A -85,B 0,C 180,E1 8613.126,E2 8613.126} C_VEL
LIN {X 0,Y 232.311,Z 825.288,A -85,B 0,C 180,E1 8609.887,E2 8609.887} C_VEL
LIN {X 0,Y 221.373,Z 839.712,A -85,B 0,C 180,E1 8606.202,E2 8606.202} C_VEL
LIN {X 0,Y 209.814,Z 854.234,A -85,B 0,C 180,E1 8601.396,E2 8601.396} C_VEL
LIN {X 0,Y 199.845,Z 866.585,A -85,B 0,C 180,E1 8596.087,E2 8596.087} C_VEL
LIN {X 0,Y 191.307,Z 877.621,A -85,B 0,C 180,E1 8590,E2 8590} C_VEL
LIN {X 0,Y 184.604,Z 887.196,A -85,B 0,C 180,E1 8583.16,E2 8583.16} C_VEL
LIN {X 0,Y 180.241,Z 894.752,A -85,B 0,C 180,E1 8575.988,E2 8575.988} C_VEL
LIN {X 0,Y 178.045,Z 900.76,A -85,B 0,C 180,E1 8568.364,E2 8568.364} C_VEL
LIN {X 0,Y 177.698,Z 904.28,A -85,B 0,C 180,E1 8562.013,E2 8562.013} C_VEL
LIN {X 0,Y 178.149,Z 906.423,A -85,B 0,C 180,E1 8555.795,E2 8555.795} C_VEL
LIN {X 0,Y 178.473,Z 907.006,A -85,B 0,C 180,E1 8550.96,E2 8550.96} C_VEL
LIN {X 0,Y 178.35,Z 906.618,A -85,B 0,C 180,E1 8546.292,E2 8546.292} C_VEL
LIN {X 0,Y 177.922,Z 905.173,A -85,B 0,C 180,E1 8541.27,E2 8541.27} C_VEL
LIN {X 0,Y 177.785,Z 902.461,A -85,B 0,C 180,E1 8535.67,E2 8535.67} C_VEL
LIN {X 0,Y 178.735,Z 897.468,A -85,B 0,C 180,E1 8528.674,E2 8528.674} C_VEL
LIN {X 0,Y 181.134,Z 891.379,A -85,B 0,C 180,E1 8522.372,E2 8522.372} C_VEL
LIN {X 0,Y 185.447,Z 883.259,A -85,B 0,C 180,E1 8515.89,E2 8515.89} C_VEL
LIN {X 0,Y 191.661,Z 873.359,A -85,B 0,C 180,E1 8509.69,E2 8509.69} C_VEL
LIN {X 0,Y 199.288,Z 861.918,A -85,B 0,C 180,E1 8504.152,E2 8504.152} C_VEL
LIN {X 0,Y 207.973,Z 849.163,A -85,B 0,C 180,E1 8499.279,E2 8499.279} C_VEL
LIN {X 0,Y 217.364,Z 835.19,A -85,B 0,C 180,E1 8495.033,E2 8495.033} C_VEL
LIN {X 0,Y 227.163,Z 819.741,A -85,B 0,C 180,E1 8491.358,E2 8491.358} C_VEL
LIN {X 0,Y 237.122,Z 802.911,A -85,B 0,C 180,E1 8488.182,E2 8488.182} C_VEL
LIN {X 0,Y 246.755,Z 785.188,A -85,B 0,C 180,E1 8485.518,E2 8485.518} C_VEL
LIN {X 0,Y 255.826,Z 766.518,A -85,B 0,C 180,E1 8483.293,E2 8483.293} C_VEL
LIN {X 0,Y 264.253,Z 746.659,A -85,B 0,C 180,E1 8481.437,E2 8481.437} C_VEL
LIN {X 0,Y 271.746,Z 726.184,A -85,B 0,C 180,E1 8479.93,E2 8479.93} C_VEL
LIN {X 0,Y 278.118,Z 705.426,A -85,B 0,C 180,E1 8478.741,E2 8478.741} C_VEL
LIN {X 0,Y 283.336,Z 683.91,A -85,B 0,C 180,E1 8477.829,E2 8477.829} C_VEL
LIN {X 0,Y 287.41,Z 661.018,A -85,B 0,C 180,E1 8477.107,E2 8477.107} C_VEL
LIN {X 0,Y 289.891,Z 637.939,A -85,B 0,C 180,E1 8476.55,E2 8476.55} C_VEL
LIN {X 0,Y 305.631,Z 446.008,A -85,B 0,C 180,E1 8472.595,E2 8472.595} C_VEL
LIN {X 0,Y 305.967,Z 441.004,A -85,B 0,C 180,E1 8472.456,E2 8472.456} C_VEL
LIN {X 0,Y 298.833,Z 429.721,A -85,B 0,C 180,E1 8468.951,E2 8468.951} C_VEL
LIN {X 0,Y 292.527,Z 420.304,A -85,B 0,C 180,E1 8465.394,E2 8465.394} C_VEL
LIN {X 0,Y 286.489,Z 411.852,A -85,B 0,C 180,E1 8461.401,E2 8461.401} C_VEL
LIN {X 0,Y 282.135,Z 406.298,A -85,B 0,C 180,E1 8458.021,E2 8458.021} C_VEL
LIN {X 0,Y 279.091,Z 402.338,A -85,B 0,C 180,E1 8455.161,E2 8455.161} C_VEL
LIN {X 0,Y 275.318,Z 397.654,A -85,B 0,C 180,E1 8450.806,E2 8450.806} C_VEL
LIN {X 0,Y 271.183,Z 393.114,A -85,B 0,C 180,E1 8442.625,E2 8442.625} C_VEL
LIN {X 0,Y 270.403,Z 392.962,A -85,B 0,C 180,E1 8438.723,E2 8438.723} C_VEL
LIN {X 0,Y 271.644,Z 396.634,A -85,B 0,C 180,E1 8430.206,E2 8430.206} C_VEL
LIN {X 0,Y 274.201,Z 401.806,A -85,B 0,C 180,E1 8425.133,E2 8425.133} C_VEL
LIN {X 0,Y 276.673,Z 406.495,A -85,B 0,C 180,E1 8421.761,E2 8421.761} C_VEL
LIN {X 0,Y 280.296,Z 412.823,A -85,B 0,C 180,E1 8418.024,E2 8418.024} C_VEL
LIN {X 0,Y 285.349,Z 422.313,A -85,B 0,C 180,E1 8413.796,E2 8413.796} C_VEL
LIN {X 0,Y 290.682,Z 432.843,A -85,B 0,C 180,E1 8410.092,E2 8410.092} C_VEL
LIN {X 0,Y 292.651,Z 437.266,A -85,B 0,C 180,E1 8408.847,E2 8408.847} C_VEL
LIN {X 0,Y 291.638,Z 479.102,A -85,B 0,C 180,E1 8406.54,E2 8406.54} C_VEL
LIN {X 0,Y 275.324,Z 638.983,A -85,B 0,C 180,E1 8403.016,E2 8403.016} C_VEL
LIN {X 0,Y 271.884,Z 660.321,A -85,B 0,C 180,E1 8402.328,E2 8402.328} C_VEL
LIN {X 0,Y 267.365,Z 680.727,A -85,B 0,C 180,E1 8401.385,E2 8401.385} C_VEL
LIN {X 0,Y 261.796,Z 700.565,A -85,B 0,C 180,E1 8400.15,E2 8400.15} C_VEL
LIN {X 0,Y 255.115,Z 720.1,A -85,B 0,C 180,E1 8398.567,E2 8398.567} C_VEL
LIN {X 0,Y 247.604,Z 738.69,A -85,B 0,C 180,E1 8396.633,E2 8396.633} C_VEL
LIN {X 0,Y 239.728,Z 755.685,A -85,B 0,C 180,E1 8394.39,E2 8394.39} C_VEL
LIN {X 0,Y 231.434,Z 771.597,A -85,B 0,C 180,E1 8391.746,E2 8391.746} C_VEL
LIN {X 0,Y 222.376,Z 787.21,A -85,B 0,C 180,E1 8388.435,E2 8388.435} C_VEL
LIN {X 0,Y 213.557,Z 801.106,A -85,B 0,C 180,E1 8384.647,E2 8384.647} C_VEL
LIN {X 0,Y 205.297,Z 813.236,A -85,B 0,C 180,E1 8380.384,E2 8380.384} C_VEL
LIN {X 0,Y 197.936,Z 823.588,A -85,B 0,C 180,E1 8375.671,E2 8375.671} C_VEL
LIN {X 0,Y 191.734,Z 832.152,A -85,B 0,C 180,E1 8370.601,E2 8370.601} C_VEL
LIN {X 0,Y 186.485,Z 839.552,A -85,B 0,C 180,E1 8364.774,E2 8364.774} C_VEL
LIN {X 0,Y 182.811,Z 845.161,A -85,B 0,C 180,E1 8358.648,E2 8358.648} C_VEL
LIN {X 0,Y 180.7,Z 848.958,A -85,B 0,C 180,E1 8352.618,E2 8352.618} C_VEL
LIN {X 0,Y 179.833,Z 851.364,A -85,B 0,C 180,E1 8346.058,E2 8346.058} C_VEL
LIN {X 0,Y 180.196,Z 852.106,A -85,B 0,C 180,E1 8339.677,E2 8339.677} C_VEL
LIN {X 0,Y 181.875,Z 851.328,A -85,B 0,C 180,E1 8333.19,E2 8333.19} C_VEL
LIN {X 0,Y 185.215,Z 848.891,A -85,B 0,C 180,E1 8326.723,E2 8326.723} C_VEL
LIN {X 0,Y 190.126,Z 844.903,A -85,B 0,C 180,E1 8320.699,E2 8320.699} C_VEL
LIN {X 0,Y 196.689,Z 839.3,A -85,B 0,C 180,E1 8315.058,E2 8315.058} C_VEL
LIN {X 0,Y 204.936,Z 831.746,A -85,B 0,C 180,E1 8309.729,E2 8309.729} C_VEL
LIN {X 0,Y 214.147,Z 822.733,A -85,B 0,C 180,E1 8305.078,E2 8305.078} C_VEL
LIN {X 0,Y 223.929,Z 812.434,A -85,B 0,C 180,E1 8301.07,E2 8301.07} C_VEL
LIN {X 0,Y 234.926,Z 799.846,A -85,B 0,C 180,E1 8297.332,E2 8297.332} C_VEL
LIN {X 0,Y 245.538,Z 786.444,A -85,B 0,C 180,E1 8294.278,E2 8294.278} C_VEL
LIN {X 0,Y 256.203,Z 771.491,A -85,B 0,C 180,E1 8291.621,E2 8291.621} C_VEL
LIN {X 0,Y 266.503,Z 755.07,A -85,B 0,C 180,E1 8289.368,E2 8289.368} C_VEL
LIN {X 0,Y 276.022,Z 737.639,A -85,B 0,C 180,E1 8287.492,E2 8287.492} C_VEL
LIN {X 0,Y 284.492,Z 719.634,A -85,B 0,C 180,E1 8285.976,E2 8285.976} C_VEL
LIN {X 0,Y 292.123,Z 700.31,A -85,B 0,C 180,E1 8284.711,E2 8284.711} C_VEL
LIN {X 0,Y 298.331,Z 681.049,A -85,B 0,C 180,E1 8283.745,E2 8283.745} C_VEL
LIN {X 0,Y 303.417,Z 660.444,A -85,B 0,C 180,E1 8282.984,E2 8282.984} C_VEL
LIN {X 0,Y 307.08,Z 639.457,A -85,B 0,C 180,E1 8282.44,E2 8282.44} C_VEL
LIN {X 0,Y 323.606,Z 503.816,A -85,B 0,C 180,E1 8279.734,E2 8279.734} C_VEL
LIN {X 0,Y 324.295,Z 497.365,A -85,B 0,C 180,E1 8279.462,E2 8279.462} C_VEL
LIN {X 0,Y 325.04,Z 488.29,A -85,B 0,C 180,E1 8278.698,E2 8278.698} C_VEL
LIN {X 0,Y 326.128,Z 475.39,A -85,B 0,C 180,E1 8277.443,E2 8277.443} C_VEL
LIN {X 0,Y 326.576,Z 471.185,A -85,B 0,C 180,E1 8277.155,E2 8277.155} C_VEL
LIN {X 0,Y 327.159,Z 466.041,A -85,B 0,C 180,E1 8276.846,E2 8276.846} C_VEL
LIN {X 0,Y 327.121,Z 463.104,A -85,B 0,C 180,E1 8274.562,E2 8274.562} C_VEL
LIN {X 0,Y 327.749,Z 461.38,A -85,B 0,C 180,E1 8271.932,E2 8271.932} C_VEL
LIN {X 0,Y 328.231,Z 461.732,A -85,B 0,C 180,E1 8270.708,E2 8270.708} C_VEL
LIN {X 0,Y 328.497,Z 462.721,A -85,B 0,C 180,E1 8270.014,E2 8270.014} C_VEL
LIN {X 0,Y 310.808,Z 619.986,A -85,B 0,C 180,E1 8266.955,E2 8266.955} C_VEL
LIN {X 0,Y 306.841,Z 653.446,A -85,B 0,C 180,E1 8266.266,E2 8266.266} C_VEL
LIN {X 0,Y 302.517,Z 675.673,A -85,B 0,C 180,E1 8265.692,E2 8265.692} C_VEL
LIN {X 0,Y 296.504,Z 697.639,A -85,B 0,C 180,E1 8264.95,E2 8264.95} C_VEL
LIN {X 0,Y 289.437,Z 718.077,A -85,B 0,C 180,E1 8264.014,E2 8264.014} C_VEL
LIN {X 0,Y 281.021,Z 738.333,A -85,B 0,C 180,E1 8262.797,E2 8262.797} C_VEL
LIN {X 0,Y 271.808,Z 757.338,A -85,B 0,C 180,E1 8261.334,E2 8261.334} C_VEL
LIN {X 0,Y 261.893,Z 775.067,A -85,B 0,C 180,E1 8259.59,E2 8259.59} C_VEL
LIN {X 0,Y 250.386,Z 793.522,A -85,B 0,C 180,E1 8257.279,E2 8257.279} C_VEL
LIN {X 0,Y 238.618,Z 810.561,A -85,B 0,C 180,E1 8254.547,E2 8254.547} C_VEL
LIN {X 0,Y 226.547,Z 826.477,A -85,B 0,C 180,E1 8251.244,E2 8251.244} C_VEL
LIN {X 0,Y 214.2,Z 841.729,A -85,B 0,C 180,E1 8247.157,E2 8247.157} C_VEL
LIN {X 0,Y 202.902,Z 855.154,A -85,B 0,C 180,E1 8242.496,E2 8242.496} C_VEL
LIN {X 0,Y 192.578,Z 867.21,A -85,B 0,C 180,E1 8237.055,E2 8237.055} C_VEL
LIN {X 0,Y 183.713,Z 877.862,A -85,B 0,C 180,E1 8230.771,E2 8230.771} C_VEL
LIN {X 0,Y 176.757,Z 887.113,A -85,B 0,C 180,E1 8223.662,E2 8223.662} C_VEL
LIN {X 0,Y 172.407,Z 894.176,A -85,B 0,C 180,E1 8216.519,E2 8216.519} C_VEL
LIN {X 0,Y 170.146,Z 899.774,A -85,B 0,C 180,E1 8208.853,E2 8208.853} C_VEL
LIN {X 0,Y 169.756,Z 903.379,A -85,B 0,C 180,E1 8201.893,E2 8201.893} C_VEL
LIN {X 0,Y 170.277,Z 905.297,A -85,B 0,C 180,E1 8195.387,E2 8195.387} C_VEL
LIN {X 0,Y 170.578,Z 905.756,A -85,B 0,C 180,E1 8190.668,E2 8190.668} C_VEL
LIN {X 0,Y 170.412,Z 905.305,A -85,B 0,C 180,E1 8185.909,E2 8185.909} C_VEL
LIN {X 0,Y 169.969,Z 903.859,A -85,B 0,C 180,E1 8180.858,E2 8180.858} C_VEL
LIN {X 0,Y 169.865,Z 901.029,A -85,B 0,C 180,E1 8174.872,E2 8174.872} C_VEL
LIN {X 0,Y 171.018,Z 895.998,A -85,B 0,C 180,E1 8167.661,E2 8167.661} C_VEL
LIN {X 0,Y 173.91,Z 889.509,A -85,B 0,C 180,E1 8160.742,E2 8160.742} C_VEL
LIN {X 0,Y 178.766,Z 881.146,A -85,B 0,C 180,E1 8154.032,E2 8154.032} C_VEL
LIN {X 0,Y 185.834,Z 870.623,A -85,B 0,C 180,E1 8147.487,E2 8147.487} C_VEL
LIN {X 0,Y 193.88,Z 859.384,A -85,B 0,C 180,E1 8142.041,E2 8142.041} C_VEL
LIN {X 0,Y 203.168,Z 846.28,A -85,B 0,C 180,E1 8137.127,E2 8137.127} C_VEL
LIN {X 0,Y 213.766,Z 830.955,A -85,B 0,C 180,E1 8132.652,E2 8132.652} C_VEL
LIN {X 0,Y 223.744,Z 815.721,A -85,B 0,C 180,E1 8129.151,E2 8129.151} C_VEL
LIN {X 0,Y 233.756,Z 799.071,A -85,B 0,C 180,E1 8126.141,E2 8126.141} C_VEL
LIN {X 0,Y 243.371,Z 781.46,A -85,B 0,C 180,E1 8123.623,E2 8123.623} C_VEL
LIN {X 0,Y 252.531,Z 762.771,A -85,B 0,C 180,E1 8121.491,E2 8121.491} C_VEL
LIN {X 0,Y 261.225,Z 742.416,A -85,B 0,C 180,E1 8119.676,E2 8119.676} C_VEL
LIN {X 0,Y 268.52,Z 722.25,A -85,B 0,C 180,E1 8118.278,E2 8118.278} C_VEL
LIN {X 0,Y 275.132,Z 700.201,A -85,B 0,C 180,E1 8117.1,E2 8117.1} C_VEL
LIN {X 0,Y 280.298,Z 678.498,A -85,B 0,C 180,E1 8116.243,E2 8116.243} C_VEL
LIN {X 0,Y 283.935,Z 656.55,A -85,B 0,C 180,E1 8115.605,E2 8115.605} C_VEL
LIN {X 0,Y 286.935,Z 624.48,A -85,B 0,C 180,E1 8114.893,E2 8114.893} C_VEL
LIN {X 0,Y 302.109,Z 445.737,A -85,B 0,C 180,E1 8111.231,E2 8111.231} C_VEL
LIN {X 0,Y 295.377,Z 434.927,A -85,B 0,C 180,E1 8107.734,E2 8107.734} C_VEL
LIN {X 0,Y 289.232,Z 425.822,A -85,B 0,C 180,E1 8104.064,E2 8104.064} C_VEL
LIN {X 0,Y 284.291,Z 418.758,A -85,B 0,C 180,E1 8100.605,E2 8100.605} C_VEL
LIN {X 0,Y 280.498,Z 413.795,A -85,B 0,C 180,E1 8097.549,E2 8097.549} C_VEL
LIN {X 0,Y 277.578,Z 409.947,A -85,B 0,C 180,E1 8094.731,E2 8094.731} C_VEL
LIN {X 0,Y 274.07,Z 405.473,A -85,B 0,C 180,E1 8090.552,E2 8090.552} C_VEL
LIN {X 0,Y 270.106,Z 401.037,A -85,B 0,C 180,E1 8082.553,E2 8082.553} C_VEL
LIN {X 0,Y 269.355,Z 400.907,A -85,B 0,C 180,E1 8078.71,E2 8078.71} C_VEL
LIN {X 0,Y 270.52,Z 404.656,A -85,B 0,C 180,E1 8070.297,E2 8070.297} C_VEL
LIN {X 0,Y 272.866,Z 409.532,A -85,B 0,C 180,E1 8065.476,E2 8065.476} C_VEL
LIN {X 0,Y 275.243,Z 414.183,A -85,B 0,C 180,E1 8062.128,E2 8062.128} C_VEL
LIN {X 0,Y 278.656,Z 420.368,A -85,B 0,C 180,E1 8058.479,E2 8058.479} C_VEL
LIN {X 0,Y 283.426,Z 429.624,A -85,B 0,C 180,E1 8054.33,E2 8054.33} C_VEL
LIN {X 0,Y 288.394,Z 439.789,A -85,B 0,C 180,E1 8050.739,E2 8050.739} C_VEL
LIN {X 0,Y 289.38,Z 442.131,A -85,B 0,C 180,E1 8050.071,E2 8050.071} C_VEL
LIN {X 0,Y 288.241,Z 480.398,A -85,B 0,C 180,E1 8047.958,E2 8047.958} C_VEL
LIN {X 0,Y 271.558,Z 639.751,A -85,B 0,C 180,E1 8044.489,E2 8044.489} C_VEL
LIN {X 0,Y 267.986,Z 661.213,A -85,B 0,C 180,E1 8043.8,E2 8043.8} C_VEL
LIN {X 0,Y 263.211,Z 682.055,A -85,B 0,C 180,E1 8042.84,E2 8042.84} C_VEL
LIN {X 0,Y 257.492,Z 701.727,A -85,B 0,C 180,E1 8041.618,E2 8041.618} C_VEL
LIN {X 0,Y 250.266,Z 722.085,A -85,B 0,C 180,E1 8039.963,E2 8039.963} C_VEL
LIN {X 0,Y 242.212,Z 741.176,A -85,B 0,C 180,E1 8037.948,E2 8037.948} C_VEL
LIN {X 0,Y 233.428,Z 759.191,A -85,B 0,C 180,E1 8035.5,E2 8035.5} C_VEL
LIN {X 0,Y 224.442,Z 775.475,A -85,B 0,C 180,E1 8032.668,E2 8032.668} C_VEL
LIN {X 0,Y 215.701,Z 789.799,A -85,B 0,C 180,E1 8029.499,E2 8029.499} C_VEL
LIN {X 0,Y 206.613,Z 803.452,A -85,B 0,C 180,E1 8025.637,E2 8025.637} C_VEL
LIN {X 0,Y 198.234,Z 815.221,A -85,B 0,C 180,E1 8021.348,E2 8021.348} C_VEL
LIN {X 0,Y 190.375,Z 825.731,A -85,B 0,C 180,E1 8016.335,E2 8016.335} C_VEL
LIN {X 0,Y 183.502,Z 834.733,A -85,B 0,C 180,E1 8010.628,E2 8010.628} C_VEL
LIN {X 0,Y 178.459,Z 841.464,A -85,B 0,C 180,E1 8004.86,E2 8004.86} C_VEL
LIN {X 0,Y 174.733,Z 846.871,A -85,B 0,C 180,E1 7998.45,E2 7998.45} C_VEL
LIN {X 0,Y 172.582,Z 850.631,A -85,B 0,C 180,E1 7991.773,E2 7991.773} C_VEL
LIN {X 0,Y 171.9,Z 852.757,A -85,B 0,C 180,E1 7985.141,E2 7985.141} C_VEL
LIN {X 0,Y 172.498,Z 853.399,A -85,B 0,C 180,E1 7978.433,E2 7978.433} C_VEL
LIN {X 0,Y 174.666,Z 852.373,A -85,B 0,C 180,E1 7971.399,E2 7971.399} C_VEL
LIN {X 0,Y 178.436,Z 849.783,A -85,B 0,C 180,E1 7964.911,E2 7964.911} C_VEL
LIN {X 0,Y 184.127,Z 845.474,A -85,B 0,C 180,E1 7958.566,E2 7958.566} C_VEL
LIN {X 0,Y 191.969,Z 839.137,A -85,B 0,C 180,E1 7952.442,E2 7952.442} C_VEL
LIN {X 0,Y 201.057,Z 831.265,A -85,B 0,C 180,E1 7947.113,E2 7947.113} C_VEL
LIN {X 0,Y 211.049,Z 821.974,A -85,B 0,C 180,E1 7942.517,E2 7942.517} C_VEL
LIN {X 0,Y 222.251,Z 810.624,A -85,B 0,C 180,E1 7938.344,E2 7938.344} C_VEL
LIN {X 0,Y 234.103,Z 797.3,A -85,B 0,C 180,E1 7934.685,E2 7934.685} C_VEL
LIN {X 0,Y 245.278,Z 783.283,A -85,B 0,C 180,E1 7931.76,E2 7931.76} C_VEL
LIN {X 0,Y 256.288,Z 767.791,A -85,B 0,C 180,E1 7929.257,E2 7929.257} C_VEL
LIN {X 0,Y 267.115,Z 750.479,A -85,B 0,C 180,E1 7927.095,E2 7927.095} C_VEL
LIN {X 0,Y 276.575,Z 732.968,A -85,B 0,C 180,E1 7925.393,E2 7925.393} C_VEL
LIN {X 0,Y 284.927,Z 714.973,A -85,B 0,C 180,E1 7924.024,E2 7924.024} C_VEL
LIN {X 0,Y 292.315,Z 695.612,A -85,B 0,C 180,E1 7922.885,E2 7922.885} C_VEL
LIN {X 0,Y 298.468,Z 675.49,A -85,B 0,C 180,E1 7921.99,E2 7921.99} C_VEL
LIN {X 0,Y 303.349,Z 654.327,A -85,B 0,C 180,E1 7921.308,E2 7921.308} C_VEL
LIN {X 0,Y 306.847,Z 631.899,A -85,B 0,C 180,E1 7920.8,E2 7920.8} C_VEL
LIN {X 0,Y 325.046,Z 485.044,A -85,B 0,C 180,E1 7917.928,E2 7917.928} C_VEL
LIN {X 0,Y 326.576,Z 471.185,A -85,B 0,C 180,E1 7917.155,E2 7917.155} C_VEL
LIN {X 0,Y 326.741,Z 469.239,A -85,B 0,C 180,E1 7916.871,E2 7916.871} C_VEL
LIN {X 0,Y 326.734,Z 468.074,A -85,B 0,C 180,E1 7916.314,E2 7916.314} C_VEL
LIN {X 0,Y 326.542,Z 468.112,A -85,B 0,C 180,E1 7915.415,E2 7915.415} C_VEL
LIN {X 0,Y 326.248,Z 470.055,A -85,B 0,C 180,E1 7913.411,E2 7913.411} C_VEL
LIN {X 0,Y 326.348,Z 469.932,A -85,B 0,C 180,E1 7912.948,E2 7912.948} C_VEL
LIN {X 0,Y 326.77,Z 469.331,A -85,B 0,C 180,E1 7911.731,E2 7911.731} C_VEL
LIN {X 0,Y 326.906,Z 469.611,A -85,B 0,C 180,E1 7911.28,E2 7911.28} C_VEL
LIN {X 0,Y 309.038,Z 623.063,A -85,B 0,C 180,E1 7908.355,E2 7908.355} C_VEL
LIN {X 0,Y 305.078,Z 654.153,A -85,B 0,C 180,E1 7907.722,E2 7907.722} C_VEL
LIN {X 0,Y 300.647,Z 676.032,A -85,B 0,C 180,E1 7907.17,E2 7907.17} C_VEL
LIN {X 0,Y 294.753,Z 697.011,A -85,B 0,C 180,E1 7906.486,E2 7906.486} C_VEL
LIN {X 0,Y 287.641,Z 717.056,A -85,B 0,C 180,E1 7905.608,E2 7905.608} C_VEL
LIN {X 0,Y 279.152,Z 737.086,A -85,B 0,C 180,E1 7904.461,E2 7904.461} C_VEL
LIN {X 0,Y 269.662,Z 756.149,A -85,B 0,C 180,E1 7903.052,E2 7903.052} C_VEL
LIN {X 0,Y 258.706,Z 775.159,A -85,B 0,C 180,E1 7901.233,E2 7901.233} C_VEL
LIN {X 0,Y 246.88,Z 793.382,A -85,B 0,C 180,E1 7898.982,E2 7898.982} C_VEL
LIN {X 0,Y 234.742,Z 810.254,A -85,B 0,C 180,E1 7896.307,E2 7896.307} C_VEL
LIN {X 0,Y 222.854,Z 825.271,A -85,B 0,C 180,E1 7893.225,E2 7893.225} C_VEL
LIN {X 0,Y 210.374,Z 840.013,A -85,B 0,C 180,E1 7889.338,E2 7889.338} C_VEL
LIN {X 0,Y 198.403,Z 853.488,A -85,B 0,C 180,E1 7884.72,E2 7884.72} C_VEL
LIN {X 0,Y 187.368,Z 865.554,A -85,B 0,C 180,E1 7879.262,E2 7879.262} C_VEL
LIN {X 0,Y 177.735,Z 876.265,A -85,B 0,C 180,E1 7872.893,E2 7872.893} C_VEL
LIN {X 0,Y 170.272,Z 885.284,A -85,B 0,C 180,E1 7865.868,E2 7865.868} C_VEL
LIN {X 0,Y 165.28,Z 892.359,A -85,B 0,C 180,E1 7858.544,E2 7858.544} C_VEL
LIN {X 0,Y 162.459,Z 898.127,A -85,B 0,C 180,E1 7850.533,E2 7850.533} C_VEL
LIN {X 0,Y 161.793,Z 901.683,A -85,B 0,C 180,E1 7843.578,E2 7843.578} C_VEL
LIN {X 0,Y 162.201,Z 903.887,A -85,B 0,C 180,E1 7836.722,E2 7836.722} C_VEL
LIN {X 0,Y 162.648,Z 904.521,A -85,B 0,C 180,E1 7831.405,E2 7831.405} C_VEL
LIN {X 0,Y 162.569,Z 904.247,A -85,B 0,C 180,E1 7826.823,E2 7826.823} C_VEL
LIN {X 0,Y 162.092,Z 902.927,A -85,B 0,C 180,E1 7821.483,E2 7821.483} C_VEL
LIN {X 0,Y 161.913,Z 900.283,A -85,B 0,C 180,E1 7815.33,E2 7815.33} C_VEL
LIN {X 0,Y 162.953,Z 895.606,A -85,B 0,C 180,E1 7807.9,E2 7807.9} C_VEL
LIN {X 0,Y 165.79,Z 889.349,A -85,B 0,C 180,E1 7800.754,E2 7800.754} C_VEL
LIN {X 0,Y 171.017,Z 880.837,A -85,B 0,C 180,E1 7793.388,E2 7793.388} C_VEL
LIN {X 0,Y 177.917,Z 871.153,A -85,B 0,C 180,E1 7786.936,E2 7786.936} C_VEL
LIN {X 0,Y 186.224,Z 859.991,A -85,B 0,C 180,E1 7781.26,E2 7781.26} C_VEL
LIN {X 0,Y 195.774,Z 847.223,A -85,B 0,C 180,E1 7776.198,E2 7776.198} C_VEL
LIN {X 0,Y 206.017,Z 833.212,A -85,B 0,C 180,E1 7771.857,E2 7771.857} C_VEL
LIN {X 0,Y 216.595,Z 817.719,A -85,B 0,C 180,E1 7768.147,E2 7768.147} C_VEL
LIN {X 0,Y 227.231,Z 800.816,A -85,B 0,C 180,E1 7764.978,E2 7764.978} C_VEL
LIN {X 0,Y 237.45,Z 782.991,A -85,B 0,C 180,E1 7762.35,E2 7762.35} C_VEL
LIN {X 0,Y 247.105,Z 764.088,A -85,B 0,C 180,E1 7760.154,E2 7760.154} C_VEL
LIN {X 0,Y 255.578,Z 744.953,A -85,B 0,C 180,E1 7758.428,E2 7758.428} C_VEL
LIN {X 0,Y 263.432,Z 724.292,A -85,B 0,C 180,E1 7756.963,E2 7756.963} C_VEL
LIN {X 0,Y 269.965,Z 703.772,A -85,B 0,C 180,E1 7755.835,E2 7755.835} C_VEL
LIN {X 0,Y 275.441,Z 681.885,A -85,B 0,C 180,E1 7754.95,E2 7754.95} C_VEL
LIN {X 0,Y 279.461,Z 659.809,A -85,B 0,C 180,E1 7754.283,E2 7754.283} C_VEL
LIN {X 0,Y 282.098,Z 635.966,A -85,B 0,C 180,E1 7753.722,E2 7753.722} C_VEL
LIN {X 0,Y 298.289,Z 450.378,A -85,B 0,C 180,E1 7749.941,E2 7749.941} C_VEL
LIN {X 0,Y 291.431,Z 439.343,A -85,B 0,C 180,E1 7746.155,E2 7746.155} C_VEL
LIN {X 0,Y 285.477,Z 430.379,A -85,B 0,C 180,E1 7742.309,E2 7742.309} C_VEL
LIN {X 0,Y 280.112,Z 422.781,A -85,B 0,C 180,E1 7738.158,E2 7738.158} C_VEL
LIN {X 0,Y 276.17,Z 417.653,A -85,B 0,C 180,E1 7734.391,E2 7734.391} C_VEL
LIN {X 0,Y 272.827,Z 413.291,A -85,B 0,C 180,E1 7730.296,E2 7730.296} C_VEL
LIN {X 0,Y 269.028,Z 408.96,A -85,B 0,C 180,E1 7722.481,E2 7722.481} C_VEL
LIN {X 0,Y 268.316,Z 408.826,A -85,B 0,C 180,E1 7718.811,E2 7718.811} C_VEL
LIN {X 0,Y 269.351,Z 412.509,A -85,B 0,C 180,E1 7710.539,E2 7710.539} C_VEL
LIN {X 0,Y 271.531,Z 417.236,A -85,B 0,C 180,E1 7705.838,E2 7705.838} C_VEL
LIN {X 0,Y 273.874,Z 421.971,A -85,B 0,C 180,E1 7702.435,E2 7702.435} C_VEL
LIN {X 0,Y 277.013,Z 427.912,A -85,B 0,C 180,E1 7698.936,E2 7698.936} C_VEL
LIN {X 0,Y 281.502,Z 436.908,A -85,B 0,C 180,E1 7694.881,E2 7694.881} C_VEL
LIN {X 0,Y 286.234,Z 446.937,A -85,B 0,C 180,E1 7691.332,E2 7691.332} C_VEL
LIN {X 0,Y 284.967,Z 481.564,A -85,B 0,C 180,E1 7689.407,E2 7689.407} C_VEL
LIN {X 0,Y 268.014,Z 639.956,A -85,B 0,C 180,E1 7686.012,E2 7686.012} C_VEL
LIN {X 0,Y 264.381,Z 661.36,A -85,B 0,C 180,E1 7685.34,E2 7685.34} C_VEL
LIN {X 0,Y 259.604,Z 681.844,A -85,B 0,C 180,E1 7684.419,E2 7684.419} C_VEL
LIN {X 0,Y 253.732,Z 701.692,A -85,B 0,C 180,E1 7683.215,E2 7683.215} C_VEL
LIN {X 0,Y 246.719,Z 721.141,A -85,B 0,C 180,E1 7681.677,E2 7681.677} C_VEL
LIN {X 0,Y 239.056,Z 739.155,A -85,B 0,C 180,E1 7679.852,E2 7679.852} C_VEL
LIN {X 0,Y 230.641,Z 756.348,A -85,B 0,C 180,E1 7677.639,E2 7677.639} C_VEL
LIN {X 0,Y 221.241,Z 773.233,A -85,B 0,C 180,E1 7674.856,E2 7674.856} C_VEL
LIN {X 0,Y 211.732,Z 788.481,A -85,B 0,C 180,E1 7671.616,E2 7671.616} C_VEL
LIN {X 0,Y 202.307,Z 802.222,A -85,B 0,C 180,E1 7667.847,E2 7667.847} C_VEL
LIN {X 0,Y 193.346,Z 814.327,A -85,B 0,C 180,E1 7663.546,E2 7663.546} C_VEL
LIN {X 0,Y 185.054,Z 824.956,A -85,B 0,C 180,E1 7658.609,E2 7658.609} C_VEL
LIN {X 0,Y 177.633,Z 834.204,A -85,B 0,C 180,E1 7652.907,E2 7652.907} C_VEL
LIN {X 0,Y 171.697,Z 841.671,A -85,B 0,C 180,E1 7646.665,E2 7646.665} C_VEL
LIN {X 0,Y 167.486,Z 847.361,A -85,B 0,C 180,E1 7640.034,E2 7640.034} C_VEL
LIN {X 0,Y 164.988,Z 851.344,A -85,B 0,C 180,E1 7633.232,E2 7633.232} C_VEL
LIN {X 0,Y 164.015,Z 853.771,A -85,B 0,C 180,E1 7626.12,E2 7626.12} C_VEL
LIN {X 0,Y 164.432,Z 854.603,A -85,B 0,C 180,E1 7619.289,E2 7619.289} C_VEL
LIN {X 0,Y 166.367,Z 853.995,A -85,B 0,C 180,E1 7612.197,E2 7612.197} C_VEL
LIN {X 0,Y 170.187,Z 851.764,A -85,B 0,C 180,E1 7605.176,E2 7605.176} C_VEL
LIN {X 0,Y 176.057,Z 847.783,A -85,B 0,C 180,E1 7598.403,E2 7598.403} C_VEL
LIN {X 0,Y 184.029,Z 841.918,A -85,B 0,C 180,E1 7592.059,E2 7592.059} C_VEL
LIN {X 0,Y 193.933,Z 833.984,A -85,B 0,C 180,E1 7586.23,E2 7586.23} C_VEL
LIN {X 0,Y 204.9,Z 824.413,A -85,B 0,C 180,E1 7581.256,E2 7581.256} C_VEL
LIN {X 0,Y 216.47,Z 813.334,A -85,B 0,C 180,E1 7577.049,E2 7577.049} C_VEL
LIN {X 0,Y 227.854,Z 801.313,A -85,B 0,C 180,E1 7573.61,E2 7573.61} C_VEL
LIN {X 0,Y 240.413,Z 786.548,A -85,B 0,C 180,E1 7570.413,E2 7570.413} C_VEL
LIN {X 0,Y 251.847,Z 771.387,A -85,B 0,C 180,E1 7567.909,E2 7567.909} C_VEL
LIN {X 0,Y 262.798,Z 754.902,A -85,B 0,C 180,E1 7565.807,E2 7565.807} C_VEL
LIN {X 0,Y 272.647,Z 737.761,A -85,B 0,C 180,E1 7564.103,E2 7564.103} C_VEL
LIN {X 0,Y 281.589,Z 719.47,A -85,B 0,C 180,E1 7562.69,E2 7562.69} C_VEL
LIN {X 0,Y 289.769,Z 699.434,A -85,B 0,C 180,E1 7561.495,E2 7561.495} C_VEL
LIN {X 0,Y 296.298,Z 679.583,A -85,B 0,C 180,E1 7560.6,E2 7560.6} C_VEL
LIN {X 0,Y 301.444,Z 659.196,A -85,B 0,C 180,E1 7559.924,E2 7559.924} C_VEL
LIN {X 0,Y 305.133,Z 637.755,A -85,B 0,C 180,E1 7559.424,E2 7559.424} C_VEL
LIN {X 0,Y 324.314,Z 486.577,A -85,B 0,C 180,E1 7556.542,E2 7556.542} C_VEL
LIN {X 0,Y 325.973,Z 472.532,A -85,B 0,C 180,E1 7555.734,E2 7555.734} C_VEL
LIN {X 0,Y 326.112,Z 470.706,A -85,B 0,C 180,E1 7554.016,E2 7554.016} C_VEL
LIN {X 0,Y 326.348,Z 469.932,A -85,B 0,C 180,E1 7552.948,E2 7552.948} C_VEL
LIN {X 0,Y 326.33,Z 470.763,A -85,B 0,C 180,E1 7552.578,E2 7552.578} C_VEL
LIN {X 0,Y 326.062,Z 473.439,A -85,B 0,C 180,E1 7552.279,E2 7552.279} C_VEL
LIN {X 0,Y 325.464,Z 478.325,A -85,B 0,C 180,E1 7552.132,E2 7552.132} C_VEL
LIN {X 0,Y 323.558,Z 492.484,A -85,B 0,C 180,E1 7552.265,E2 7552.265} C_VEL
LIN {X 0,Y 323.438,Z 493.425,A -85,B 0,C 180,E1 7552.251,E2 7552.251} C_VEL
LIN {X 0,Y 304.4,Z 650.507,A -85,B 0,C 180,E1 7549.292,E2 7549.292} C_VEL
LIN {X 0,Y 299.915,Z 672.93,A -85,B 0,C 180,E1 7548.761,E2 7548.761} C_VEL
LIN {X 0,Y 294.22,Z 693.328,A -85,B 0,C 180,E1 7548.146,E2 7548.146} C_VEL
LIN {X 0,Y 286.905,Z 714.145,A -85,B 0,C 180,E1 7547.317,E2 7547.317} C_VEL
LIN {X 0,Y 278.463,Z 734.055,A -85,B 0,C 180,E1 7546.263,E2 7546.263} C_VEL
LIN {X 0,Y 268.391,Z 753.874,A -85,B 0,C 180,E1 7544.883,E2 7544.883} C_VEL
LIN {X 0,Y 257.869,Z 771.926,A -85,B 0,C 180,E1 7543.268,E2 7543.268} C_VEL
LIN {X 0,Y 246.081,Z 789.855,A -85,B 0,C 180,E1 7541.201,E2 7541.201} C_VEL
LIN {X 0,Y 233.477,Z 806.956,A -85,B 0,C 180,E1 7538.653,E2 7538.653} C_VEL
LIN {X 0,Y 220.673,Z 822.665,A -85,B 0,C 180,E1 7535.597,E2 7535.597} C_VEL
LIN {X 0,Y 207.565,Z 837.581,A -85,B 0,C 180,E1 7531.82,E2 7531.82} C_VEL
LIN {X 0,Y 194.862,Z 851.205,A -85,B 0,C 180,E1 7527.293,E2 7527.293} C_VEL
LIN {X 0,Y 182.449,Z 863.94,A -85,B 0,C 180,E1 7521.592,E2 7521.592} C_VEL
LIN {X 0,Y 172.016,Z 874.685,A -85,B 0,C 180,E1 7515.159,E2 7515.159} C_VEL
LIN {X 0,Y 163.859,Z 883.683,A -85,B 0,C 180,E1 7508.041,E2 7508.041} C_VEL
LIN {X 0,Y 157.925,Z 891.18,A -85,B 0,C 180,E1 7500.006,E2 7500.006} C_VEL
LIN {X 0,Y 154.647,Z 897.029,A -85,B 0,C 180,E1 7491.403,E2 7491.403} C_VEL
LIN {X 0,Y 153.849,Z 900.631,A -85,B 0,C 180,E1 7483.91,E2 7483.91} C_VEL
LIN {X 0,Y 154.282,Z 902.706,A -85,B 0,C 180,E1 7476.695,E2 7476.695} C_VEL
LIN {X 0,Y 154.741,Z 903.274,A -85,B 0,C 180,E1 7471.477,E2 7471.477} C_VEL
LIN {X 0,Y 154.65,Z 902.972,A -85,B 0,C 180,E1 7466.66,E2 7466.66} C_VEL
LIN {X 0,Y 154.136,Z 901.604,A -85,B 0,C 180,E1 7461.04,E2 7461.04} C_VEL
LIN {X 0,Y 153.984,Z 899.086,A -85,B 0,C 180,E1 7454.942,E2 7454.942} C_VEL
LIN {X 0,Y 155.161,Z 894.416,A -85,B 0,C 180,E1 7447.147,E2 7447.147} C_VEL
LIN {X 0,Y 158.28,Z 888.142,A -85,B 0,C 180,E1 7439.641,E2 7439.641} C_VEL
LIN {X 0,Y 163.94,Z 879.601,A -85,B 0,C 180,E1 7431.972,E2 7431.972} C_VEL
LIN {X 0,Y 171.129,Z 870.119,A -85,B 0,C 180,E1 7425.465,E2 7425.465} C_VEL
LIN {X 0,Y 180.145,Z 858.668,A -85,B 0,C 180,E1 7419.508,E2 7419.508} C_VEL
LIN {X 0,Y 190.207,Z 845.826,A -85,B 0,C 180,E1 7414.377,E2 7414.377} C_VEL
LIN {X 0,Y 200.931,Z 831.678,A -85,B 0,C 180,E1 7410.016,E2 7410.016} C_VEL
LIN {X 0,Y 211.936,Z 816.119,A -85,B 0,C 180,E1 7406.31,E2 7406.31} C_VEL
LIN {X 0,Y 222.471,Z 799.872,A -85,B 0,C 180,E1 7403.298,E2 7403.298} C_VEL
LIN {X 0,Y 232.614,Z 782.676,A -85,B 0,C 180,E1 7400.784,E2 7400.784} C_VEL
LIN {X 0,Y 242.63,Z 763.531,A -85,B 0,C 180,E1 7398.587,E2 7398.587} C_VEL
LIN {X 0,Y 251.308,Z 744.399,A -85,B 0,C 180,E1 7396.885,E2 7396.885} C_VEL
LIN {X 0,Y 259.492,Z 723.329,A -85,B 0,C 180,E1 7395.419,E2 7395.419} C_VEL
LIN {X 0,Y 266.223,Z 702.468,A -85,B 0,C 180,E1 7394.303,E2 7394.303} C_VEL
LIN {X 0,Y 271.802,Z 680.518,A -85,B 0,C 180,E1 7393.442,E2 7393.442} C_VEL
LIN {X 0,Y 275.794,Z 658.674,A -85,B 0,C 180,E1 7392.802,E2 7392.802} C_VEL
LIN {X 0,Y 278.655,Z 632.34,A -85,B 0,C 180,E1 7392.201,E2 7392.201} C_VEL
LIN {X 0,Y 294.537,Z 455.068,A -85,B 0,C 180,E1 7388.618,E2 7388.618} C_VEL
LIN {X 0,Y 288.391,Z 445.075,A -85,B 0,C 180,E1 7385.023,E2 7385.023} C_VEL
LIN {X 0,Y 282.558,Z 436.218,A -85,B 0,C 180,E1 7381.015,E2 7381.015} C_VEL
LIN {X 0,Y 277.721,Z 429.372,A -85,B 0,C 180,E1 7377.008,E2 7377.008} C_VEL
LIN {X 0,Y 274.674,Z 425.248,A -85,B 0,C 180,E1 7373.941,E2 7373.941} C_VEL
LIN {X 0,Y 271.59,Z 421.109,A -85,B 0,C 180,E1 7370.037,E2 7370.037} C_VEL
LIN {X 0,Y 267.887,Z 416.817,A -85,B 0,C 180,E1 7362.179,E2 7362.179} C_VEL
LIN {X 0,Y 267.257,Z 416.805,A -85,B 0,C 180,E1 7358.683,E2 7358.683} C_VEL
LIN {X 0,Y 268.222,Z 420.491,A -85,B 0,C 180,E1 7350.66,E2 7350.66} C_VEL
LIN {X 0,Y 270.23,Z 424.996,A -85,B 0,C 180,E1 7346.163,E2 7346.163} C_VEL
LIN {X 0,Y 272.485,Z 429.705,A -85,B 0,C 180,E1 7342.777,E2 7342.777} C_VEL
LIN {X 0,Y 275.425,Z 435.548,A -85,B 0,C 180,E1 7339.354,E2 7339.354} C_VEL
LIN {X 0,Y 279.541,Z 444.066,A -85,B 0,C 180,E1 7335.49,E2 7335.49} C_VEL
LIN {X 0,Y 283.179,Z 452.06,A -85,B 0,C 180,E1 7332.595,E2 7332.595} C_VEL
LIN {X 0,Y 281.883,Z 482.715,A -85,B 0,C 180,E1 7330.889,E2 7330.889} C_VEL
LIN {X 0,Y 264.561,Z 640.745,A -85,B 0,C 180,E1 7327.558,E2 7327.558} C_VEL
LIN {X 0,Y 260.793,Z 662.266,A -85,B 0,C 180,E1 7326.89,E2 7326.89} C_VEL
LIN {X 0,Y 255.804,Z 683.001,A -85,B 0,C 180,E1 7325.967,E2 7325.967} C_VEL
LIN {X 0,Y 249.782,Z 702.72,A -85,B 0,C 180,E1 7324.782,E2 7324.782} C_VEL
LIN {X 0,Y 242.151,Z 723.144,A -85,B 0,C 180,E1 7323.171,E2 7323.171} C_VEL
LIN {X 0,Y 233.594,Z 742.351,A -85,B 0,C 180,E1 7321.195,E2 7321.195} C_VEL
LIN {X 0,Y 224.252,Z 760.414,A -85,B 0,C 180,E1 7318.788,E2 7318.788} C_VEL
LIN {X 0,Y 214.617,Z 776.79,A -85,B 0,C 180,E1 7315.974,E2 7315.974} C_VEL
LIN {X 0,Y 204.863,Z 791.656,A -85,B 0,C 180,E1 7312.682,E2 7312.682} C_VEL
LIN {X 0,Y 195.179,Z 805.105,A -85,B 0,C 180,E1 7308.831,E2 7308.831} C_VEL
LIN {X 0,Y 185.702,Z 817.281,A -85,B 0,C 180,E1 7304.274,E2 7304.274} C_VEL
LIN {X 0,Y 176.667,Z 828.241,A -85,B 0,C 180,E1 7298.793,E2 7298.793} C_VEL
LIN {X 0,Y 169.051,Z 837.203,A -85,B 0,C 180,E1 7292.716,E2 7292.716} C_VEL
LIN {X 0,Y 163.15,Z 844.243,A -85,B 0,C 180,E1 7286.138,E2 7286.138} C_VEL
LIN {X 0,Y 159.223,Z 849.299,A -85,B 0,C 180,E1 7279.511,E2 7279.511} C_VEL
LIN {X 0,Y 156.749,Z 853.186,A -85,B 0,C 180,E1 7271.878,E2 7271.878} C_VEL
LIN {X 0,Y 156.083,Z 855.274,A -85,B 0,C 180,E1 7264.583,E2 7264.583} C_VEL
LIN {X 0,Y 156.909,Z 855.925,A -85,B 0,C 180,E1 7257.21,E2 7257.21} C_VEL
LIN {X 0,Y 159.463,Z 854.975,A -85,B 0,C 180,E1 7249.778,E2 7249.778} C_VEL
LIN {X 0,Y 164.08,Z 852.387,A -85,B 0,C 180,E1 7242.501,E2 7242.501} C_VEL
LIN {X 0,Y 170.877,Z 848.049,A -85,B 0,C 180,E1 7235.584,E2 7235.584} C_VEL
LIN {X 0,Y 179.811,Z 841.828,A -85,B 0,C 180,E1 7229.197,E2 7229.197} C_VEL
LIN {X 0,Y 189.48,Z 834.522,A -85,B 0,C 180,E1 7223.972,E2 7223.972} C_VEL
LIN {X 0,Y 201.016,Z 825.012,A -85,B 0,C 180,E1 7219.091,E2 7219.091} C_VEL
LIN {X 0,Y 213.171,Z 813.869,A -85,B 0,C 180,E1 7214.947,E2 7214.947} C_VEL
LIN {X 0,Y 225.467,Z 801.355,A -85,B 0,C 180,E1 7211.481,E2 7211.481} C_VEL
LIN {X 0,Y 237.614,Z 787.528,A -85,B 0,C 180,E1 7208.582,E2 7208.582} C_VEL
LIN {X 0,Y 249.39,Z 772.479,A -85,B 0,C 180,E1 7206.158,E2 7206.158} C_VEL
LIN {X 0,Y 260.626,Z 756.131,A -85,B 0,C 180,E1 7204.128,E2 7204.128} C_VEL
LIN {X 0,Y 271.189,Z 738.263,A -85,B 0,C 180,E1 7202.413,E2 7202.413} C_VEL
LIN {X 0,Y 280.317,Z 720.071,A -85,B 0,C 180,E1 7201.064,E2 7201.064} C_VEL
LIN {X 0,Y 288.395,Z 700.788,A -85,B 0,C 180,E1 7199.956,E2 7199.956} C_VEL
LIN {X 0,Y 295.13,Z 680.94,A -85,B 0,C 180,E1 7199.089,E2 7199.089} C_VEL
LIN {X 0,Y 300.348,Z 660.895,A -85,B 0,C 180,E1 7198.442,E2 7198.442} C_VEL
LIN {X 0,Y 304.169,Z 639.85,A -85,B 0,C 180,E1 7197.96,E2 7197.96} C_VEL
LIN {X 0,Y 323.825,Z 488.148,A -85,B 0,C 180,E1 7195.151,E2 7195.151} C_VEL
LIN {X 0,Y 324.988,Z 479.195,A -85,B 0,C 180,E1 7194.615,E2 7194.615} C_VEL
LIN {X 0,Y 325.418,Z 477.769,A -85,B 0,C 180,E1 7192.539,E2 7192.539} C_VEL
LIN {X 0,Y 323.438,Z 493.425,A -85,B 0,C 180,E1 7192.251,E2 7192.251} C_VEL
LIN {X 0,Y 322.417,Z 501.123,A -85,B 0,C 180,E1 7192.289,E2 7192.289} C_VEL
LIN {X 0,Y 319.531,Z 521.76,A -85,B 0,C 180,E1 7193.034,E2 7193.034} C_VEL
LIN {X 0,Y 318.661,Z 528.361,A -85,B 0,C 180,E1 7193.047,E2 7193.047} C_VEL
LIN {X 0,Y 303.467,Z 649.915,A -85,B 0,C 180,E1 7190.806,E2 7190.806} C_VEL
LIN {X 0,Y 298.845,Z 672.378,A -85,B 0,C 180,E1 7190.296,E2 7190.296} C_VEL
LIN {X 0,Y 292.916,Z 693.151,A -85,B 0,C 180,E1 7189.7,E2 7189.7} C_VEL
LIN {X 0,Y 285.286,Z 714.267,A -85,B 0,C 180,E1 7188.897,E2 7188.897} C_VEL
LIN {X 0,Y 276.709,Z 733.849,A -85,B 0,C 180,E1 7187.902,E2 7187.902} C_VEL
LIN {X 0,Y 266.242,Z 753.941,A -85,B 0,C 180,E1 7186.559,E2 7186.559} C_VEL
LIN {X 0,Y 255.183,Z 772.2,A -85,B 0,C 180,E1 7184.969,E2 7184.969} C_VEL
LIN {X 0,Y 242.437,Z 790.797,A -85,B 0,C 180,E1 7182.859,E2 7182.859} C_VEL
LIN {X 0,Y 229.332,Z 807.826,A -85,B 0,C 180,E1 7180.335,E2 7180.335} C_VEL
LIN {X 0,Y 215.768,Z 823.687,A -85,B 0,C 180,E1 7177.235,E2 7177.235} C_VEL
LIN {X 0,Y 202.238,Z 838.219,A -85,B 0,C 180,E1 7173.483,E2 7173.483} C_VEL
LIN {X 0,Y 189.063,Z 851.513,A -85,B 0,C 180,E1 7168.945,E2 7168.945} C_VEL
LIN {X 0,Y 176.687,Z 863.495,A -85,B 0,C 180,E1 7163.466,E2 7163.466} C_VEL
LIN {X 0,Y 165.629,Z 874.067,A -85,B 0,C 180,E1 7156.918,E2 7156.918} C_VEL
LIN {X 0,Y 156.182,Z 883.622,A -85,B 0,C 180,E1 7148.852,E2 7148.852} C_VEL
LIN {X 0,Y 150.002,Z 890.935,A -85,B 0,C 180,E1 7140.432,E2 7140.432} C_VEL
LIN {X 0,Y 146.782,Z 896.134,A -85,B 0,C 180,E1 7131.998,E2 7131.998} C_VEL
LIN {X 0,Y 145.902,Z 899.837,A -85,B 0,C 180,E1 7123.469,E2 7123.469} C_VEL
LIN {X 0,Y 146.361,Z 901.526,A -85,B 0,C 180,E1 7116.665,E2 7116.665} C_VEL
LIN {X 0,Y 146.833,Z 902.022,A -85,B 0,C 180,E1 7111.557,E2 7111.557} C_VEL
LIN {X 0,Y 146.757,Z 901.756,A -85,B 0,C 180,E1 7106.872,E2 7106.872} C_VEL
LIN {X 0,Y 146.206,Z 900.399,A -85,B 0,C 180,E1 7100.946,E2 7100.946} C_VEL
LIN {X 0,Y 146.062,Z 897.885,A -85,B 0,C 180,E1 7094.512,E2 7094.512} C_VEL
LIN {X 0,Y 147.393,Z 893.23,A -85,B 0,C 180,E1 7086.321,E2 7086.321} C_VEL
LIN {X 0,Y 150.834,Z 886.911,A -85,B 0,C 180,E1 7078.416,E2 7078.416} C_VEL
LIN {X 0,Y 156.981,Z 878.318,A -85,B 0,C 180,E1 7070.417,E2 7070.417} C_VEL
LIN {X 0,Y 164.663,Z 868.831,A -85,B 0,C 180,E1 7063.727,E2 7063.727} C_VEL
LIN {X 0,Y 174.243,Z 857.304,A -85,B 0,C 180,E1 7057.633,E2 7057.633} C_VEL
LIN {X 0,Y 184.847,Z 844.367,A -85,B 0,C 180,E1 7052.449,E2 7052.449} C_VEL
LIN {X 0,Y 196.057,Z 830.127,A -85,B 0,C 180,E1 7048.078,E2 7048.078} C_VEL
LIN {X 0,Y 206.982,Z 815.199,A -85,B 0,C 180,E1 7044.548,E2 7044.548} C_VEL
LIN {X 0,Y 217.969,Z 798.714,A -85,B 0,C 180,E1 7041.53,E2 7041.53} C_VEL
LIN {X 0,Y 228.919,Z 780.528,A -85,B 0,C 180,E1 7038.935,E2 7038.935} C_VEL
LIN {X 0,Y 238.832,Z 761.997,A -85,B 0,C 180,E1 7036.866,E2 7036.866} C_VEL
LIN {X 0,Y 247.654,Z 742.868,A -85,B 0,C 180,E1 7035.214,E2 7035.214} C_VEL
LIN {X 0,Y 255.736,Z 722.304,A -85,B 0,C 180,E1 7033.831,E2 7033.831} C_VEL
LIN {X 0,Y 262.456,Z 701.754,A -85,B 0,C 180,E1 7032.764,E2 7032.764} C_VEL
LIN {X 0,Y 268.062,Z 680.051,A -85,B 0,C 180,E1 7031.936,E2 7031.936} C_VEL
LIN {X 0,Y 272.1,Z 658.297,A -85,B 0,C 180,E1 7031.313,E2 7031.313} C_VEL
LIN {X 0,Y 275.069,Z 631.562,A -85,B 0,C 180,E1 7030.71,E2 7030.71} C_VEL
LIN {X 0,Y 290.968,Z 459.892,A -85,B 0,C 180,E1 7027.28,E2 7027.28} C_VEL
LIN {X 0,Y 284.636,Z 449.517,A -85,B 0,C 180,E1 7023.323,E2 7023.323} C_VEL
LIN {X 0,Y 279.34,Z 441.465,A -85,B 0,C 180,E1 7019.385,E2 7019.385} C_VEL
LIN {X 0,Y 275.591,Z 436.205,A -85,B 0,C 180,E1 7016.048,E2 7016.048} C_VEL
LIN {X 0,Y 273.174,Z 432.835,A -85,B 0,C 180,E1 7013.486,E2 7013.486} C_VEL
LIN {X 0,Y 270.308,Z 428.892,A -85,B 0,C 180,E1 7009.721,E2 7009.721} C_VEL
LIN {X 0,Y 266.812,Z 424.739,A -85,B 0,C 180,E1 7002.105,E2 7002.105} C_VEL
LIN {X 0,Y 266.204,Z 424.771,A -85,B 0,C 180,E1 6998.635,E2 6998.635} C_VEL
LIN {X 0,Y 267.068,Z 428.371,A -85,B 0,C 180,E1 6990.877,E2 6990.877} C_VEL
LIN {X 0,Y 268.939,Z 432.756,A -85,B 0,C 180,E1 6986.491,E2 6986.491} C_VEL
LIN {X 0,Y 271.048,Z 437.349,A -85,B 0,C 180,E1 6983.179,E2 6983.179} C_VEL
LIN {X 0,Y 273.928,Z 443.348,A -85,B 0,C 180,E1 6979.694,E2 6979.694} C_VEL
LIN {X 0,Y 277.629,Z 451.298,A -85,B 0,C 180,E1 6976.08,E2 6976.08} C_VEL
LIN {X 0,Y 280.227,Z 457.428,A -85,B 0,C 180,E1 6973.867,E2 6973.867} C_VEL
LIN {X 0,Y 278.922,Z 483.915,A -85,B 0,C 180,E1 6972.396,E2 6972.396} C_VEL
LIN {X 0,Y 261.349,Z 641.01,A -85,B 0,C 180,E1 6969.154,E2 6969.154} C_VEL
LIN {X 0,Y 257.502,Z 662.556,A -85,B 0,C 180,E1 6968.502,E2 6968.502} C_VEL
LIN {X 0,Y 252.368,Z 683.449,A -85,B 0,C 180,E1 6967.594,E2 6967.594} C_VEL
LIN {X 0,Y 246.022,Z 703.707,A -85,B 0,C 180,E1 6966.398,E2 6966.398} C_VEL
LIN {X 0,Y 238.582,Z 723.149,A -85,B 0,C 180,E1 6964.896,E2 6964.896} C_VEL
LIN {X 0,Y 230.259,Z 741.517,A -85,B 0,C 180,E1 6963.066,E2 6963.066} C_VEL
LIN {X 0,Y 221.418,Z 758.443,A -85,B 0,C 180,E1 6960.912,E2 6960.912} C_VEL
LIN {X 0,Y 211.566,Z 775.016,A -85,B 0,C 180,E1 6958.206,E2 6958.206} C_VEL
LIN {X 0,Y 201.344,Z 790.283,A -85,B 0,C 180,E1 6954.97,E2 6954.97} C_VEL
LIN {X 0,Y 191.133,Z 804.051,A -85,B 0,C 180,E1 6951.162,E2 6951.162} C_VEL
LIN {X 0,Y 181.732,Z 815.71,A -85,B 0,C 180,E1 6946.957,E2 6946.957} C_VEL
LIN {X 0,Y 172.312,Z 826.711,A -85,B 0,C 180,E1 6941.721,E2 6941.721} C_VEL
LIN {X 0,Y 163.724,Z 836.344,A -85,B 0,C 180,E1 6935.493,E2 6935.493} C_VEL
LIN {X 0,Y 157.009,Z 843.868,A -85,B 0,C 180,E1 6928.773,E2 6928.773} C_VEL
LIN {X 0,Y 152.272,Z 849.525,A -85,B 0,C 180,E1 6921.698,E2 6921.698} C_VEL
LIN {X 0,Y 149.316,Z 853.67,A -85,B 0,C 180,E1 6914.069,E2 6914.069} C_VEL
LIN {X 0,Y 148.206,Z 856.071,A -85,B 0,C 180,E1 6906.549,E2 6906.549} C_VEL
LIN {X 0,Y 148.676,Z 857.101,A -85,B 0,C 180,E1 6898.818,E2 6898.818} C_VEL
LIN {X 0,Y 151.02,Z 856.635,A -85,B 0,C 180,E1 6890.768,E2 6890.768} C_VEL
LIN {X 0,Y 155.313,Z 854.671,A -85,B 0,C 180,E1 6883.332,E2 6883.332} C_VEL
LIN {X 0,Y 162.407,Z 850.672,A -85,B 0,C 180,E1 6875.651,E2 6875.651} C_VEL
LIN {X 0,Y 171.466,Z 844.939,A -85,B 0,C 180,E1 6868.945,E2 6868.945} C_VEL
LIN {X 0,Y 181.757,Z 837.747,A -85,B 0,C 180,E1 6863.276,E2 6863.276} C_VEL
LIN {X 0,Y 193.151,Z 829.038,A -85,B 0,C 180,E1 6858.406,E2 6858.406} C_VEL
LIN {X 0,Y 206.082,Z 818.123,A -85,B 0,C 180,E1 6854.002,E2 6854.002} C_VEL
LIN {X 0,Y 218.618,Z 806.332,A -85,B 0,C 180,E1 6850.501,E2 6850.501} C_VEL
LIN {X 0,Y 231.71,Z 792.551,A -85,B 0,C 180,E1 6847.437,E2 6847.437} C_VEL
LIN {X 0,Y 243.874,Z 777.927,A -85,B 0,C 180,E1 6844.984,E2 6844.984} C_VEL
LIN {X 0,Y 255.684,Z 761.837,A -85,B 0,C 180,E1 6842.913,E2 6842.913} C_VEL
LIN {X 0,Y 267.002,Z 744.012,A -85,B 0,C 180,E1 6841.144,E2 6841.144} C_VEL
LIN {X 0,Y 276.95,Z 725.648,A -85,B 0,C 180,E1 6839.742,E2 6839.742} C_VEL
LIN {X 0,Y 285.528,Z 706.747,A -85,B 0,C 180,E1 6838.628,E2 6838.628} C_VEL
LIN {X 0,Y 292.67,Z 687.219,A -85,B 0,C 180,E1 6837.749,E2 6837.749} C_VEL
LIN {X 0,Y 298.653,Z 666.211,A -85,B 0,C 180,E1 6837.048,E2 6837.048} C_VEL
LIN {X 0,Y 302.993,Z 645.027,A -85,B 0,C 180,E1 6836.548,E2 6836.548} C_VEL
LIN {X 0,Y 323.604,Z 489.755,A -85,B 0,C 180,E1 6833.758,E2 6833.758} C_VEL
LIN {X 0,Y 318.661,Z 528.361,A -85,B 0,C 180,E1 6833.047,E2 6833.047} C_VEL
LIN {X 0,Y 318.64,Z 528.685,A -85,B 0,C 180,E1 6833.044,E2 6833.044} C_VEL
LIN {X 0,Y 318.64,Z 634.639,A -85,B 0,C 180,E1 6833.044,E2 6833.044} C_VEL
LIN {X 0,Y 315.545,Z 634.639,A -85,B 0,C 180,E1 6834.056,E2 6834.056} C_VEL
LIN {X 0,Y 314.598,Z 632.639,A -85,B 0,C 180,E1 6834.376,E2 6834.376} C_VEL
LIN {X 0,Y 314.598,Z 572.023,A -85,B 0,C 180,E1 6834.376,E2 6834.376} C_VEL
LIN {X 0,Y 312.86,Z 571.489,A -85,B 0,C 180,E1 6833.733,E2 6833.733} C_VEL
LIN {X 0,Y 302.781,Z 649.475,A -85,B 0,C 180,E1 6832.326,E2 6832.326} C_VEL
LIN {X 0,Y 297.938,Z 672.461,A -85,B 0,C 180,E1 6831.828,E2 6831.828} C_VEL
LIN {X 0,Y 291.833,Z 693.241,A -85,B 0,C 180,E1 6831.262,E2 6831.262} C_VEL
LIN {X 0,Y 284.316,Z 713.487,A -85,B 0,C 180,E1 6830.536,E2 6830.536} C_VEL
LIN {X 0,Y 275.485,Z 733.23,A -85,B 0,C 180,E1 6829.587,E2 6829.587} C_VEL
LIN {X 0,Y 264.965,Z 752.95,A -85,B 0,C 180,E1 6828.338,E2 6828.338} C_VEL
LIN {X 0,Y 253.11,Z 772.009,A -85,B 0,C 180,E1 6826.754,E2 6826.754} C_VEL
LIN {X 0,Y 239.937,Z 790.562,A -85,B 0,C 180,E1 6824.719,E2 6824.719} C_VEL
LIN {X 0,Y 226.232,Z 807.704,A -85,B 0,C 180,E1 6822.244,E2 6822.244} C_VEL
LIN {X 0,Y 211.847,Z 823.862,A -85,B 0,C 180,E1 6819.139,E2 6819.139} C_VEL
LIN {X 0,Y 197.839,Z 838.141,A -85,B 0,C 180,E1 6815.455,E2 6815.455} C_VEL
LIN {X 0,Y 183.433,Z 851.846,A -85,B 0,C 180,E1 6810.7,E2 6810.7} C_VEL
LIN {X 0,Y 170.522,Z 863.594,A -85,B 0,C 180,E1 6805.167,E2 6805.167} C_VEL
LIN {X 0,Y 158.907,Z 873.927,A -85,B 0,C 180,E1 6798.476,E2 6798.476} C_VEL
LIN {X 0,Y 149.277,Z 882.855,A -85,B 0,C 180,E1 6790.514,E2 6790.514} C_VEL
LIN {X 0,Y 142.554,Z 890.016,A -85,B 0,C 180,E1 6781.733,E2 6781.733} C_VEL
LIN {X 0,Y 138.979,Z 895.148,A -85,B 0,C 180,E1 6772.856,E2 6772.856} C_VEL
LIN {X 0,Y 137.965,Z 898.727,A -85,B 0,C 180,E1 6763.799,E2 6763.799} C_VEL
LIN {X 0,Y 138.44,Z 900.348,A -85,B 0,C 180,E1 6756.631,E2 6756.631} C_VEL
LIN {X 0,Y 138.923,Z 900.774,A -85,B 0,C 180,E1 6751.645,E2 6751.645} C_VEL
LIN {X 0,Y 138.835,Z 900.473,A -85,B 0,C 180,E1 6746.693,E2 6746.693} C_VEL
LIN {X 0,Y 138.245,Z 899.063,A -85,B 0,C 180,E1 6740.42,E2 6740.42} C_VEL
LIN {X 0,Y 138.174,Z 896.483,A -85,B 0,C 180,E1 6733.603,E2 6733.603} C_VEL
LIN {X 0,Y 139.773,Z 891.761,A -85,B 0,C 180,E1 6725.031,E2 6725.031} C_VEL
LIN {X 0,Y 143.458,Z 885.669,A -85,B 0,C 180,E1 6717.064,E2 6717.064} C_VEL
LIN {X 0,Y 149.975,Z 877.226,A -85,B 0,C 180,E1 6708.883,E2 6708.883} C_VEL
LIN {X 0,Y 158.374,Z 867.477,A -85,B 0,C 180,E1 6701.839,E2 6701.839} C_VEL
LIN {X 0,Y 168.541,Z 855.915,A -85,B 0,C 180,E1 6695.63,E2 6695.63} C_VEL
LIN {X 0,Y 179.051,Z 843.675,A -85,B 0,C 180,E1 6690.682,E2 6690.682} C_VEL
LIN {X 0,Y 190.702,Z 829.433,A -85,B 0,C 180,E1 6686.285,E2 6686.285} C_VEL
LIN {X 0,Y 202.549,Z 813.788,A -85,B 0,C 180,E1 6682.61,E2 6682.61} C_VEL
LIN {X 0,Y 213.688,Z 797.541,A -85,B 0,C 180,E1 6679.688,E2 6679.688} C_VEL
LIN {X 0,Y 224.965,Z 779.232,A -85,B 0,C 180,E1 6677.137,E2 6677.137} C_VEL
LIN {X 0,Y 235.112,Z 760.565,A -85,B 0,C 180,E1 6675.117,E2 6675.117} C_VEL
LIN {X 0,Y 244.208,Z 741.151,A -85,B 0,C 180,E1 6673.497,E2 6673.497} C_VEL
LIN {X 0,Y 252.142,Z 721.214,A -85,B 0,C 180,E1 6672.202,E2 6672.202} C_VEL
LIN {X 0,Y 259.104,Z 700.125,A -85,B 0,C 180,E1 6671.148,E2 6671.148} C_VEL
LIN {X 0,Y 264.894,Z 677.941,A -85,B 0,C 180,E1 6670.336,E2 6670.336} C_VEL
LIN {X 0,Y 268.902,Z 655.931,A -85,B 0,C 180,E1 6669.732,E2 6669.732} C_VEL
LIN {X 0,Y 272.225,Z 624.849,A -85,B 0,C 180,E1 6669.06,E2 6669.06} C_VEL
LIN {X 0,Y 287.393,Z 464.712,A -85,B 0,C 180,E1 6665.891,E2 6665.891} C_VEL
LIN {X 0,Y 282.185,Z 456.076,A -85,B 0,C 180,E1 6662.438,E2 6662.438} C_VEL
LIN {X 0,Y 277.465,Z 448.692,A -85,B 0,C 180,E1 6658.762,E2 6658.762} C_VEL
LIN {X 0,Y 273.934,Z 443.618,A -85,B 0,C 180,E1 6655.5,E2 6655.5} C_VEL
LIN {X 0,Y 271.686,Z 440.419,A -85,B 0,C 180,E1 6653.025,E2 6653.025} C_VEL
LIN {X 0,Y 269.092,Z 436.738,A -85,B 0,C 180,E1 6649.511,E2 6649.511} C_VEL
LIN {X 0,Y 265.737,Z 432.661,A -85,B 0,C 180,E1 6642.03,E2 6642.03} C_VEL
LIN {X 0,Y 265.147,Z 432.711,A -85,B 0,C 180,E1 6638.663,E2 6638.663} C_VEL
LIN {X 0,Y 265.913,Z 436.224,A -85,B 0,C 180,E1 6631.121,E2 6631.121} C_VEL
LIN {X 0,Y 267.667,Z 440.543,A -85,B 0,C 180,E1 6626.801,E2 6626.801} C_VEL
LIN {X 0,Y 269.686,Z 445.123,A -85,B 0,C 180,E1 6623.498,E2 6623.498} C_VEL
LIN {X 0,Y 272.382,Z 451.006,A -85,B 0,C 180,E1 6620.105,E2 6620.105} C_VEL
LIN {X 0,Y 275.75,Z 458.562,A -85,B 0,C 180,E1 6616.67,E2 6616.67} C_VEL
LIN {X 0,Y 277.402,Z 462.6,A -85,B 0,C 180,E1 6615.178,E2 6615.178} C_VEL
LIN {X 0,Y 276.151,Z 485.072,A -85,B 0,C 180,E1 6613.935,E2 6613.935} C_VEL
LIN {X 0,Y 258.224,Z 641.862,A -85,B 0,C 180,E1 6610.77,E2 6610.77} C_VEL
LIN {X 0,Y 254.221,Z 663.607,A -85,B 0,C 180,E1 6610.123,E2 6610.123} C_VEL
LIN {X 0,Y 248.974,Z 684.339,A -85,B 0,C 180,E1 6609.238,E2 6609.238} C_VEL
LIN {X 0,Y 242.494,Z 704.475,A -85,B 0,C 180,E1 6608.073,E2 6608.073} C_VEL
LIN {X 0,Y 234.538,Z 724.653,A -85,B 0,C 180,E1 6606.536,E2 6606.536} C_VEL
LIN {X 0,Y 225.393,Z 744.068,A -85,B 0,C 180,E1 6604.601,E2 6604.601} C_VEL
LIN {X 0,Y 215.48,Z 762.117,A -85,B 0,C 180,E1 6602.253,E2 6602.253} C_VEL
LIN {X 0,Y 205.196,Z 778.505,A -85,B 0,C 180,E1 6599.484,E2 6599.484} C_VEL
LIN {X 0,Y 194.708,Z 793.399,A -85,B 0,C 180,E1 6596.211,E2 6596.211} C_VEL
LIN {X 0,Y 184.212,Z 806.891,A -85,B 0,C 180,E1 6592.333,E2 6592.333} C_VEL
LIN {X 0,Y 173.958,Z 818.975,A -85,B 0,C 180,E1 6587.739,E2 6587.739} C_VEL
LIN {X 0,Y 164.305,Z 829.584,A -85,B 0,C 180,E1 6582.301,E2 6582.301} C_VEL
LIN {X 0,Y 156.069,Z 838.275,A -85,B 0,C 180,E1 6576.256,E2 6576.256} C_VEL
LIN {X 0,Y 149.131,Z 845.61,A -85,B 0,C 180,E1 6569.236,E2 6569.236} C_VEL
LIN {X 0,Y 143.976,Z 851.447,A -85,B 0,C 180,E1 6561.216,E2 6561.216} C_VEL
LIN {X 0,Y 141.12,Z 855.365,A -85,B 0,C 180,E1 6553.031,E2 6553.031} C_VEL
LIN {X 0,Y 140.267,Z 857.656,A -85,B 0,C 180,E1 6544.857,E2 6544.857} C_VEL
LIN {X 0,Y 141.165,Z 858.429,A -85,B 0,C 180,E1 6536.694,E2 6536.694} C_VEL
LIN {X 0,Y 144.031,Z 857.727,A -85,B 0,C 180,E1 6528.564,E2 6528.564} C_VEL
LIN {X 0,Y 149.487,Z 855.326,A -85,B 0,C 180,E1 6520.322,E2 6520.322} C_VEL
LIN {X 0,Y 157.181,Z 851.273,A -85,B 0,C 180,E1 6512.902,E2 6512.902} C_VEL
LIN {X 0,Y 166.925,Z 845.541,A -85,B 0,C 180,E1 6506.31,E2 6506.31} C_VEL
LIN {X 0,Y 178.312,Z 838.044,A -85,B 0,C 180,E1 6500.551,E2 6500.551} C_VEL
LIN {X 0,Y 190.996,Z 828.739,A -85,B 0,C 180,E1 6495.598,E2 6495.598} C_VEL
LIN {X 0,Y 204.068,Z 818.029,A -85,B 0,C 180,E1 6491.517,E2 6491.517} C_VEL
LIN {X 0,Y 217.6,Z 805.628,A -85,B 0,C 180,E1 6488.05,E2 6488.05} C_VEL
LIN {X 0,Y 230.902,Z 791.886,A -85,B 0,C 180,E1 6485.193,E2 6485.193} C_VEL
LIN {X 0,Y 243.266,Z 777.449,A -85,B 0,C 180,E1 6482.912,E2 6482.912} C_VEL
LIN {X 0,Y 254.99,Z 761.684,A -85,B 0,C 180,E1 6481.008,E2 6481.008} C_VEL
LIN {X 0,Y 266.431,Z 744.004,A -85,B 0,C 180,E1 6479.354,E2 6479.354} C_VEL
LIN {X 0,Y 276.101,Z 726.526,A -85,B 0,C 180,E1 6478.09,E2 6478.09} C_VEL
LIN {X 0,Y 285.262,Z 706.721,A -85,B 0,C 180,E1 6476.986,E2 6476.986} C_VEL
LIN {X 0,Y 292.346,Z 687.655,A -85,B 0,C 180,E1 6476.175,E2 6476.175} C_VEL
LIN {X 0,Y 298.447,Z 666.632,A -85,B 0,C 180,E1 6475.511,E2 6475.511} C_VEL
LIN {X 0,Y 302.846,Z 645.53,A -85,B 0,C 180,E1 6475.037,E2 6475.037} C_VEL
LIN {X 0,Y 312.86,Z 571.489,A -85,B 0,C 180,E1 6473.733,E2 6473.733} C_VEL
LIN {X 0,Y 316.124,Z 571.808,A -85,B 0,C 180,E1 6473.32,E2 6473.32} C_VEL
LIN {X 0,Y 316.124,Z 687.985,A -85,B 0,C 180,E1 6473.32,E2 6473.32} C_VEL
LIN {X 0,Y 304.802,Z 687.985,A -85,B 0,C 180,E1 6474.208,E2 6474.208} C_VEL
LIN {X 0,Y 302.969,Z 685.985,A -85,B 0,C 180,E1 6474.359,E2 6474.359} C_VEL
LIN {X 0,Y 302.969,Z 656.79,A -85,B 0,C 180,E1 6474.359,E2 6474.359} C_VEL
LIN {X 0,Y 301.051,Z 656.088,A -85,B 0,C 180,E1 6473.721,E2 6473.721} C_VEL
LIN {X 0,Y 295.637,Z 678.524,A -85,B 0,C 180,E1 6473.228,E2 6473.228} C_VEL
LIN {X 0,Y 289.016,Z 699.062,A -85,B 0,C 180,E1 6472.661,E2 6472.661} C_VEL
LIN {X 0,Y 281.22,Z 718.502,A -85,B 0,C 180,E1 6471.947,E2 6471.947} C_VEL
LIN {X 0,Y 271.927,Z 737.687,A -85,B 0,C 180,E1 6471.013,E2 6471.013} C_VEL
LIN {X 0,Y 260.157,Z 758.298,A -85,B 0,C 180,E1 6469.683,E2 6469.683} C_VEL
LIN {X 0,Y 248.17,Z 776.439,A -85,B 0,C 180,E1 6468.142,E2 6468.142} C_VEL
LIN {X 0,Y 233.897,Z 795.298,A -85,B 0,C 180,E1 6466.006,E2 6466.006} C_VEL
LIN {X 0,Y 219.606,Z 811.859,A -85,B 0,C 180,E1 6463.489,E2 6463.489} C_VEL
LIN {X 0,Y 204.883,Z 827.285,A -85,B 0,C 180,E1 6460.357,E2 6460.357} C_VEL
LIN {X 0,Y 189.804,Z 841.711,A -85,B 0,C 180,E1 6456.399,E2 6456.399} C_VEL
LIN {X 0,Y 175.163,Z 854.705,A -85,B 0,C 180,E1 6451.52,E2 6451.52} C_VEL
LIN {X 0,Y 161.418,Z 866.212,A -85,B 0,C 180,E1 6445.463,E2 6445.463} C_VEL
LIN {X 0,Y 149.242,Z 876.302,A -85,B 0,C 180,E1 6438.037,E2 6438.037} C_VEL
LIN {X 0,Y 139.707,Z 884.659,A -85,B 0,C 180,E1 6429.38,E2 6429.38} C_VEL
LIN {X 0,Y 133.532,Z 890.975,A -85,B 0,C 180,E1 6420.106,E2 6420.106} C_VEL
LIN {X 0,Y 130.466,Z 895.648,A -85,B 0,C 180,E1 6410.169,E2 6410.169} C_VEL
LIN {X 0,Y 130.088,Z 898.313,A -85,B 0,C 180,E1 6401.523,E2 6401.523} C_VEL
LIN {X 0,Y 130.821,Z 899.49,A -85,B 0,C 180,E1 6393.94,E2 6393.94} C_VEL
LIN {X 0,Y 131.043,Z 899.475,A -85,B 0,C 180,E1 6388.684,E2 6388.684} C_VEL
LIN {X 0,Y 130.539,Z 898.581,A -85,B 0,C 180,E1 6382.956,E2 6382.956} C_VEL
LIN {X 0,Y 130.17,Z 896.202,A -85,B 0,C 180,E1 6375.312,E2 6375.312} C_VEL
LIN {X 0,Y 131.178,Z 892.366,A -85,B 0,C 180,E1 6367.12,E2 6367.12} C_VEL
LIN {X 0,Y 134.896,Z 886.107,A -85,B 0,C 180,E1 6357.671,E2 6357.671} C_VEL
LIN {X 0,Y 141.045,Z 878.492,A -85,B 0,C 180,E1 6349.289,E2 6349.289} C_VEL
LIN {X 0,Y 149.728,Z 868.815,A -85,B 0,C 180,E1 6341.584,E2 6341.584} C_VEL
LIN {X 0,Y 160.048,Z 857.706,A -85,B 0,C 180,E1 6335.071,E2 6335.071} C_VEL
LIN {X 0,Y 171.405,Z 845.247,A -85,B 0,C 180,E1 6329.632,E2 6329.632} C_VEL
LIN {X 0,Y 183.34,Z 831.399,A -85,B 0,C 180,E1 6325.131,E2 6325.131} C_VEL
LIN {X 0,Y 195.059,Z 816.654,A -85,B 0,C 180,E1 6321.503,E2 6321.503} C_VEL
LIN {X 0,Y 207.091,Z 800.041,A -85,B 0,C 180,E1 6318.373,E2 6318.373} C_VEL
LIN {X 0,Y 218.729,Z 782.119,A -85,B 0,C 180,E1 6315.788,E2 6315.788} C_VEL
LIN {X 0,Y 229.499,Z 763.095,A -85,B 0,C 180,E1 6313.693,E2 6313.693} C_VEL
LIN {X 0,Y 238.786,Z 744.243,A -85,B 0,C 180,E1 6312.086,E2 6312.086} C_VEL
LIN {X 0,Y 246.873,Z 725.182,A -85,B 0,C 180,E1 6310.81,E2 6310.81} C_VEL
LIN {X 0,Y 254.213,Z 704.175,A -85,B 0,C 180,E1 6309.738,E2 6309.738} C_VEL
LIN {X 0,Y 260.156,Z 682.805,A -85,B 0,C 180,E1 6308.933,E2 6308.933} C_VEL
LIN {X 0,Y 264.869,Z 659.669,A -85,B 0,C 180,E1 6308.276,E2 6308.276} C_VEL
LIN {X 0,Y 267.748,Z 636.903,A -85,B 0,C 180,E1 6307.759,E2 6307.759} C_VEL
LIN {X 0,Y 284.038,Z 469.683,A -85,B 0,C 180,E1 6304.498,E2 6304.498} C_VEL
LIN {X 0,Y 278.505,Z 460.386,A -85,B 0,C 180,E1 6300.515,E2 6300.515} C_VEL
LIN {X 0,Y 273.804,Z 453.068,A -85,B 0,C 180,E1 6296.442,E2 6296.442} C_VEL
LIN {X 0,Y 270.392,Z 448.234,A -85,B 0,C 180,E1 6292.778,E2 6292.778} C_VEL
LIN {X 0,Y 267.694,Z 444.413,A -85,B 0,C 180,E1 6289.02,E2 6289.02} C_VEL
LIN {X 0,Y 264.663,Z 440.582,A -85,B 0,C 180,E1 6281.955,E2 6281.955} C_VEL
LIN {X 0,Y 264.085,Z 440.663,A -85,B 0,C 180,E1 6278.656,E2 6278.656} C_VEL
LIN {X 0,Y 264.768,Z 444.102,A -85,B 0,C 180,E1 6271.342,E2 6271.342} C_VEL
LIN {X 0,Y 266.383,Z 448.273,A -85,B 0,C 180,E1 6267.156,E2 6267.156} C_VEL
LIN {X 0,Y 268.344,Z 452.921,A -85,B 0,C 180,E1 6263.803,E2 6263.803} C_VEL
LIN {X 0,Y 270.802,Z 458.548,A -85,B 0,C 180,E1 6260.577,E2 6260.577} C_VEL
LIN {X 0,Y 273.859,Z 465.737,A -85,B 0,C 180,E1 6257.301,E2 6257.301} C_VEL
LIN {X 0,Y 274.66,Z 467.948,A -85,B 0,C 180,E1 6256.5,E2 6256.5} C_VEL
LIN {X 0,Y 273.524,Z 486.264,A -85,B 0,C 180,E1 6255.5,E2 6255.5} C_VEL
LIN {X 0,Y 255.352,Z 642.276,A -85,B 0,C 180,E1 6252.434,E2 6252.434} C_VEL
LIN {X 0,Y 251.255,Z 664.075,A -85,B 0,C 180,E1 6251.805,E2 6251.805} C_VEL
LIN {X 0,Y 245.973,Z 684.542,A -85,B 0,C 180,E1 6250.958,E2 6250.958} C_VEL
LIN {X 0,Y 239.549,Z 704.192,A -85,B 0,C 180,E1 6249.862,E2 6249.862} C_VEL
LIN {X 0,Y 231.456,Z 724.416,A -85,B 0,C 180,E1 6248.379,E2 6248.379} C_VEL
LIN {X 0,Y 222.4,Z 743.354,A -85,B 0,C 180,E1 6246.565,E2 6246.565} C_VEL
LIN {X 0,Y 212.564,Z 761.023,A -85,B 0,C 180,E1 6244.367,E2 6244.367} C_VEL
LIN {X 0,Y 202.246,Z 777.249,A -85,B 0,C 180,E1 6241.755,E2 6241.755} C_VEL
LIN {X 0,Y 190.992,Z 792.896,A -85,B 0,C 180,E1 6238.453,E2 6238.453} C_VEL
LIN {X 0,Y 179.998,Z 806.585,A -85,B 0,C 180,E1 6234.624,E2 6234.624} C_VEL
LIN {X 0,Y 169.177,Z 818.841,A -85,B 0,C 180,E1 6230.05,E2 6230.05} C_VEL
LIN {X 0,Y 159.248,Z 829.31,A -85,B 0,C 180,E1 6224.787,E2 6224.787} C_VEL
LIN {X 0,Y 150.05,Z 838.564,A -85,B 0,C 180,E1 6218.434,E2 6218.434} C_VEL
LIN {X 0,Y 142.477,Z 846.101,A -85,B 0,C 180,E1 6211.21,E2 6211.21} C_VEL
LIN {X 0,Y 136.97,Z 851.894,A -85,B 0,C 180,E1 6203.297,E2 6203.297} C_VEL
LIN {X 0,Y 133.605,Z 856.068,A -85,B 0,C 180,E1 6194.82,E2 6194.82} C_VEL
LIN {X 0,Y 132.366,Z 858.593,A -85,B 0,C 180,E1 6186.06,E2 6186.06} C_VEL
LIN {X 0,Y 133.108,Z 859.637,A -85,B 0,C 180,E1 6177.274,E2 6177.274} C_VEL
LIN {X 0,Y 136.224,Z 859.146,A -85,B 0,C 180,E1 6168.099,E2 6168.099} C_VEL
LIN {X 0,Y 141.717,Z 857.075,A -85,B 0,C 180,E1 6159.741,E2 6159.741} C_VEL
LIN {X 0,Y 149.986,Z 853.189,A -85,B 0,C 180,E1 6151.777,E2 6151.777} C_VEL
LIN {X 0,Y 160.791,Z 847.32,A -85,B 0,C 180,E1 6144.62,E2 6144.62} C_VEL
LIN {X 0,Y 173.054,Z 839.774,A -85,B 0,C 180,E1 6138.653,E2 6138.653} C_VEL
LIN {X 0,Y 186.276,Z 830.642,A -85,B 0,C 180,E1 6133.718,E2 6133.718} C_VEL
LIN {X 0,Y 199.812,Z 820.179,A -85,B 0,C 180,E1 6129.694,E2 6129.694} C_VEL
LIN {X 0,Y 213.748,Z 808.068,A -85,B 0,C 180,E1 6126.301,E2 6126.301} C_VEL
LIN {X 0,Y 227.385,Z 794.694,A -85,B 0,C 180,E1 6123.526,E2 6123.526} C_VEL
LIN {X 0,Y 241.001,Z 779.357,A -85,B 0,C 180,E1 6121.151,E2 6121.151} C_VEL
LIN {X 0,Y 253.07,Z 763.763,A -85,B 0,C 180,E1 6119.32,E2 6119.32} C_VEL
LIN {X 0,Y 265.165,Z 745.679,A -85,B 0,C 180,E1 6117.688,E2 6117.688} C_VEL
LIN {X 0,Y 275.479,Z 727.59,A -85,B 0,C 180,E1 6116.439,E2 6116.439} C_VEL
LIN {X 0,Y 284.345,Z 708.903,A -85,B 0,C 180,E1 6115.442,E2 6115.442} C_VEL
LIN {X 0,Y 291.975,Z 689.036,A -85,B 0,C 180,E1 6114.632,E2 6114.632} C_VEL
LIN {X 0,Y 298.321,Z 667.834,A -85,B 0,C 180,E1 6113.992,E2 6113.992} C_VEL
LIN {X 0,Y 301.051,Z 656.088,A -85,B 0,C 180,E1 6113.721,E2 6113.721} C_VEL
LIN {X 0,Y 304.582,Z 656.533,A -85,B 0,C 180,E1 6113.386,E2 6113.386} C_VEL
LIN {X 0,Y 304.582,Z 727.059,A -85,B 0,C 180,E1 6113.386,E2 6113.386} C_VEL
LIN {X 0,Y 289.243,Z 727.059,A -85,B 0,C 180,E1 6114.073,E2 6114.073} C_VEL
LIN {X 0,Y 287.298,Z 725.059,A -85,B 0,C 180,E1 6114.165,E2 6114.165} C_VEL
LIN {X 0,Y 287.298,Z 711.822,A -85,B 0,C 180,E1 6114.165,E2 6114.165} C_VEL
LIN {X 0,Y 283.766,Z 710.974,A -85,B 0,C 180,E1 6113.878,E2 6113.878} C_VEL
LIN {X 0,Y 274.468,Z 731.087,A -85,B 0,C 180,E1 6113.044,E2 6113.044} C_VEL
LIN {X 0,Y 263.542,Z 750.777,A -85,B 0,C 180,E1 6111.956,E2 6111.956} C_VEL
LIN {X 0,Y 251.687,Z 769.084,A -85,B 0,C 180,E1 6110.625,E2 6110.625} C_VEL
LIN {X 0,Y 238.041,Z 787.491,A -85,B 0,C 180,E1 6108.859,E2 6108.859} C_VEL
LIN {X 0,Y 224.392,Z 803.767,A -85,B 0,C 180,E1 6106.792,E2 6106.792} C_VEL
LIN {X 0,Y 209.896,Z 819.099,A -85,B 0,C 180,E1 6104.193,E2 6104.193} C_VEL
LIN {X 0,Y 194.175,Z 834.131,A -85,B 0,C 180,E1 6100.757,E2 6100.757} C_VEL
LIN {X 0,Y 178.772,Z 847.602,A -85,B 0,C 180,E1 6096.516,E2 6096.516} C_VEL
LIN {X 0,Y 163.799,Z 859.776,A -85,B 0,C 180,E1 6091.168,E2 6091.168} C_VEL
LIN {X 0,Y 150.095,Z 870.325,A -85,B 0,C 180,E1 6084.58,E2 6084.58} C_VEL
LIN {X 0,Y 138.157,Z 879.549,A -85,B 0,C 180,E1 6076.355,E2 6076.355} C_VEL
LIN {X 0,Y 129.424,Z 886.861,A -85,B 0,C 180,E1 6067.049,E2 6067.049} C_VEL
LIN {X 0,Y 124.083,Z 892.326,A -85,B 0,C 180,E1 6056.818,E2 6056.818} C_VEL
LIN {X 0,Y 122.107,Z 896.119,A -85,B 0,C 180,E1 6046.16,E2 6046.16} C_VEL
LIN {X 0,Y 122.386,Z 897.731,A -85,B 0,C 180,E1 6038.451,E2 6038.451} C_VEL
LIN {X 0,Y 123.022,Z 898.256,A -85,B 0,C 180,E1 6032.79,E2 6032.79} C_VEL
LIN {X 0,Y 123.115,Z 898.153,A -85,B 0,C 180,E1 6028.134,E2 6028.134} C_VEL
LIN {X 0,Y 122.526,Z 897.144,A -85,B 0,C 180,E1 6022.021,E2 6022.021} C_VEL
LIN {X 0,Y 122.283,Z 894.598,A -85,B 0,C 180,E1 6013.854,E2 6013.854} C_VEL
LIN {X 0,Y 123.829,Z 890.386,A -85,B 0,C 180,E1 6004.658,E2 6004.658} C_VEL
LIN {X 0,Y 128.094,Z 884.179,A -85,B 0,C 180,E1 5995.258,E2 5995.258} C_VEL
LIN {X 0,Y 135.182,Z 876.203,A -85,B 0,C 180,E1 5986.458,E2 5986.458} C_VEL
LIN {X 0,Y 144.725,Z 866.403,A -85,B 0,C 180,E1 5978.672,E2 5978.672} C_VEL
LIN {X 0,Y 155.895,Z 854.964,A -85,B 0,C 180,E1 5972.15,E2 5972.15} C_VEL
LIN {X 0,Y 168.022,Z 842.151,A -85,B 0,C 180,E1 5966.79,E2 5966.79} C_VEL
LIN {X 0,Y 180.597,Z 827.934,A -85,B 0,C 180,E1 5962.388,E2 5962.388} C_VEL
LIN {X 0,Y 193.273,Z 812.276,A -85,B 0,C 180,E1 5958.781,E2 5958.781} C_VEL
LIN {X 0,Y 205.258,Z 795.78,A -85,B 0,C 180,E1 5955.912,E2 5955.912} C_VEL
LIN {X 0,Y 216.975,Z 777.687,A -85,B 0,C 180,E1 5953.503,E2 5953.503} C_VEL
LIN {X 0,Y 227.612,Z 758.939,A -85,B 0,C 180,E1 5951.584,E2 5951.584} C_VEL
LIN {X 0,Y 237.116,Z 739.428,A -85,B 0,C 180,E1 5950.054,E2 5950.054} C_VEL
LIN {X 0,Y 245.385,Z 719.264,A -85,B 0,C 180,E1 5948.836,E2 5948.836} C_VEL
LIN {X 0,Y 252.591,Z 697.917,A -85,B 0,C 180,E1 5947.853,E2 5947.853} C_VEL
LIN {X 0,Y 258.346,Z 676.355,A -85,B 0,C 180,E1 5947.127,E2 5947.127} C_VEL
LIN {X 0,Y 262.46,Z 654.255,A -85,B 0,C 180,E1 5946.553,E2 5946.553} C_VEL
LIN {X 0,Y 266.184,Z 620.124,A -85,B 0,C 180,E1 5945.85,E2 5945.85} C_VEL
LIN {X 0,Y 280.739,Z 474.662,A -85,B 0,C 180,E1 5943.063,E2 5943.063} C_VEL
LIN {X 0,Y 275.437,Z 465.77,A -85,B 0,C 180,E1 5938.961,E2 5938.961} C_VEL
LIN {X 0,Y 271.389,Z 459.474,A -85,B 0,C 180,E1 5935.14,E2 5935.14} C_VEL
LIN {X 0,Y 268.831,Z 455.699,A -85,B 0,C 180,E1 5932.199,E2 5932.199} C_VEL
LIN {X 0,Y 266.454,Z 452.226,A -85,B 0,C 180,E1 5928.749,E2 5928.749} C_VEL
LIN {X 0,Y 263.59,Z 448.504,A -85,B 0,C 180,E1 5921.879,E2 5921.879} C_VEL
LIN {X 0,Y 263.049,Z 448.558,A -85,B 0,C 180,E1 5918.833,E2 5918.833} C_VEL
LIN {X 0,Y 263.61,Z 451.902,A -85,B 0,C 180,E1 5911.641,E2 5911.641} C_VEL
LIN {X 0,Y 265.116,Z 456.03,A -85,B 0,C 180,E1 5907.493,E2 5907.493} C_VEL
LIN {X 0,Y 267.148,Z 461.031,A -85,B 0,C 180,E1 5903.895,E2 5903.895} C_VEL
LIN {X 0,Y 269.57,Z 466.901,A -85,B 0,C 180,E1 5900.637,E2 5900.637} C_VEL
LIN {X 0,Y 272.079,Z 473.211,A -85,B 0,C 180,E1 5897.853,E2 5897.853} C_VEL
LIN {X 0,Y 271.084,Z 487.399,A -85,B 0,C 180,E1 5897.093,E2 5897.093} C_VEL
LIN {X 0,Y 252.6,Z 643,A -85,B 0,C 180,E1 5894.122,E2 5894.122} C_VEL
LIN {X 0,Y 248.314,Z 665.193,A -85,B 0,C 180,E1 5893.498,E2 5893.498} C_VEL
LIN {X 0,Y 242.762,Z 686.042,A -85,B 0,C 180,E1 5892.653,E2 5892.653} C_VEL
LIN {X 0,Y 235.946,Z 706.173,A -85,B 0,C 180,E1 5891.547,E2 5891.547} C_VEL
LIN {X 0,Y 227.95,Z 725.516,A -85,B 0,C 180,E1 5890.152,E2 5890.152} C_VEL
LIN {X 0,Y 218.433,Z 744.826,A -85,B 0,C 180,E1 5888.336,E2 5888.336} C_VEL
LIN {X 0,Y 208.336,Z 762.385,A -85,B 0,C 180,E1 5886.182,E2 5886.182} C_VEL
LIN {X 0,Y 197.756,Z 778.476,A -85,B 0,C 180,E1 5883.62,E2 5883.62} C_VEL
LIN {X 0,Y 186.83,Z 793.212,A -85,B 0,C 180,E1 5880.561,E2 5880.561} C_VEL
LIN {X 0,Y 174.692,Z 807.797,A -85,B 0,C 180,E1 5876.519,E2 5876.519} C_VEL
LIN {X 0,Y 163.414,Z 820.023,A -85,B 0,C 180,E1 5871.919,E2 5871.919} C_VEL
LIN {X 0,Y 153.205,Z 830.273,A -85,B 0,C 180,E1 5866.692,E2 5866.692} C_VEL
LIN {X 0,Y 143.298,Z 839.721,A -85,B 0,C 180,E1 5860.05,E2 5860.05} C_VEL
LIN {X 0,Y 135.091,Z 847.41,A -85,B 0,C 180,E1 5852.364,E2 5852.364} C_VEL
LIN {X 0,Y 129.363,Z 853.067,A -85,B 0,C 180,E1 5844.238,E2 5844.238} C_VEL
LIN {X 0,Y 125.758,Z 857.257,A -85,B 0,C 180,E1 5835.266,E2 5835.266} C_VEL
LIN {X 0,Y 124.459,Z 859.724,A -85,B 0,C 180,E1 5826.319,E2 5826.319} C_VEL
LIN {X 0,Y 125.238,Z 860.881,A -85,B 0,C 180,E1 5816.956,E2 5816.956} C_VEL
LIN {X 0,Y 128.511,Z 860.543,A -85,B 0,C 180,E1 5807.406,E2 5807.406} C_VEL
LIN {X 0,Y 134.355,Z 858.657,A -85,B 0,C 180,E1 5798.619,E2 5798.619} C_VEL
LIN {X 0,Y 143.352,Z 854.807,A -85,B 0,C 180,E1 5790.14,E2 5790.14} C_VEL
LIN {X 0,Y 154.305,Z 849.326,A -85,B 0,C 180,E1 5783.067,E2 5783.067} C_VEL
LIN {X 0,Y 166.953,Z 842.135,A -85,B 0,C 180,E1 5777.063,E2 5777.063} C_VEL
LIN {X 0,Y 180.926,Z 833.169,A -85,B 0,C 180,E1 5772.015,E2 5772.015} C_VEL
LIN {X 0,Y 195.181,Z 822.838,A -85,B 0,C 180,E1 5767.949,E2 5767.949} C_VEL
LIN {X 0,Y 209.631,Z 810.986,A -85,B 0,C 180,E1 5764.595,E2 5764.595} C_VEL
LIN {X 0,Y 224.141,Z 797.347,A -85,B 0,C 180,E1 5761.788,E2 5761.788} C_VEL
LIN {X 0,Y 237.46,Z 783.059,A -85,B 0,C 180,E1 5759.591,E2 5759.591} C_VEL
LIN {X 0,Y 251.164,Z 766.203,A -85,B 0,C 180,E1 5757.641,E2 5757.641} C_VEL
LIN {X 0,Y 262.523,Z 750.081,A -85,B 0,C 180,E1 5756.212,E2 5756.212} C_VEL
LIN {X 0,Y 273.424,Z 731.809,A -85,B 0,C 180,E1 5754.964,E2 5754.964} C_VEL
LIN {X 0,Y 282.488,Z 713.761,A -85,B 0,C 180,E1 5754.011,E2 5754.011} C_VEL
LIN {X 0,Y 283.766,Z 710.974,A -85,B 0,C 180,E1 5753.878,E2 5753.878} C_VEL
LIN {X 0,Y 285.859,Z 712.249,A -85,B 0,C 180,E1 5753.304,E2 5753.304} C_VEL
LIN {X 0,Y 285.859,Z 758.451,A -85,B 0,C 180,E1 5753.304,E2 5753.304} C_VEL
LIN {X 0,Y 271.357,Z 758.451,A -85,B 0,C 180,E1 5754.219,E2 5754.219} C_VEL
LIN {X 0,Y 269.451,Z 756.451,A -85,B 0,C 180,E1 5754.347,E2 5754.347} C_VEL
LIN {X 0,Y 269.451,Z 746.21,A -85,B 0,C 180,E1 5754.347,E2 5754.347} C_VEL
LIN {X 0,Y 266.071,Z 745.122,A -85,B 0,C 180,E1 5754.036,E2 5754.036} C_VEL
LIN {X 0,Y 254.885,Z 762.869,A -85,B 0,C 180,E1 5752.936,E2 5752.936} C_VEL
LIN {X 0,Y 242.107,Z 780.381,A -85,B 0,C 180,E1 5751.508,E2 5751.508} C_VEL
LIN {X 0,Y 227.683,Z 797.727,A -85,B 0,C 180,E1 5749.617,E2 5749.617} C_VEL
LIN {X 0,Y 213.124,Z 813.304,A -85,B 0,C 180,E1 5747.359,E2 5747.359} C_VEL
LIN {X 0,Y 197.253,Z 828.485,A -85,B 0,C 180,E1 5744.372,E2 5744.372} C_VEL
LIN {X 0,Y 181.233,Z 842.211,A -85,B 0,C 180,E1 5740.619,E2 5740.619} C_VEL
LIN {X 0,Y 164.651,Z 855.225,A -85,B 0,C 180,E1 5735.609,E2 5735.609} C_VEL
LIN {X 0,Y 149.581,Z 866.321,A -85,B 0,C 180,E1 5729.467,E2 5729.467} C_VEL
LIN {X 0,Y 136.14,Z 875.864,A -85,B 0,C 180,E1 5721.791,E2 5721.791} C_VEL
LIN {X 0,Y 125.468,Z 883.562,A -85,B 0,C 180,E1 5712.631,E2 5712.631} C_VEL
LIN {X 0,Y 117.957,Z 889.813,A -85,B 0,C 180,E1 5701.698,E2 5701.698} C_VEL
LIN {X 0,Y 114.626,Z 893.911,A -85,B 0,C 180,E1 5690.949,E2 5690.949} C_VEL
LIN {X 0,Y 114.284,Z 896.272,A -85,B 0,C 180,E1 5680.582,E2 5680.582} C_VEL
LIN {X 0,Y 115.046,Z 896.983,A -85,B 0,C 180,E1 5673.483,E2 5673.483} C_VEL
LIN {X 0,Y 115.231,Z 896.918,A -85,B 0,C 180,E1 5668.503,E2 5668.503} C_VEL
LIN {X 0,Y 114.645,Z 896.038,A -85,B 0,C 180,E1 5662.478,E2 5662.478} C_VEL
LIN {X 0,Y 114.353,Z 893.545,A -85,B 0,C 180,E1 5653.747,E2 5653.747} C_VEL
LIN {X 0,Y 116.019,Z 889.38,A -85,B 0,C 180,E1 5643.921,E2 5643.921} C_VEL
LIN {X 0,Y 120.622,Z 883.235,A -85,B 0,C 180,E1 5633.941,E2 5633.941} C_VEL
LIN {X 0,Y 128.169,Z 875.361,A -85,B 0,C 180,E1 5624.767,E2 5624.767} C_VEL
LIN {X 0,Y 138.377,Z 865.535,A -85,B 0,C 180,E1 5616.668,E2 5616.668} C_VEL
LIN {X 0,Y 149.483,Z 854.769,A -85,B 0,C 180,E1 5610.355,E2 5610.355} C_VEL
LIN {X 0,Y 162.685,Z 841.458,A -85,B 0,C 180,E1 5604.705,E2 5604.705} C_VEL
LIN {X 0,Y 175.093,Z 828.054,A -85,B 0,C 180,E1 5600.518,E2 5600.518} C_VEL
LIN {X 0,Y 188.143,Z 812.489,A -85,B 0,C 180,E1 5596.937,E2 5596.937} C_VEL
LIN {X 0,Y 200.472,Z 796.094,A -85,B 0,C 180,E1 5594.102,E2 5594.102} C_VEL
LIN {X 0,Y 212.429,Z 778.227,A -85,B 0,C 180,E1 5591.749,E2 5591.749} C_VEL
LIN {X 0,Y 223.286,Z 759.722,A -85,B 0,C 180,E1 5589.877,E2 5589.877} C_VEL
LIN {X 0,Y 232.948,Z 740.452,A -85,B 0,C 180,E1 5588.392,E2 5588.392} C_VEL
LIN {X 0,Y 241.401,Z 720.605,A -85,B 0,C 180,E1 5587.208,E2 5587.208} C_VEL
LIN {X 0,Y 248.727,Z 699.751,A -85,B 0,C 180,E1 5586.257,E2 5586.257} C_VEL
LIN {X 0,Y 254.813,Z 677.689,A -85,B 0,C 180,E1 5585.528,E2 5585.528} C_VEL
LIN {X 0,Y 259.041,Z 656.062,A -85,B 0,C 180,E1 5584.978,E2 5584.978} C_VEL
LIN {X 0,Y 262.519,Z 626.594,A -85,B 0,C 180,E1 5584.368,E2 5584.368} C_VEL
LIN {X 0,Y 277.574,Z 479.816,A -85,B 0,C 180,E1 5581.6,E2 5581.6} C_VEL
LIN {X 0,Y 272.916,Z 471.736,A -85,B 0,C 180,E1 5577.691,E2 5577.691} C_VEL
LIN {X 0,Y 269.383,Z 466.279,A -85,B 0,C 180,E1 5574.128,E2 5574.128} C_VEL
LIN {X 0,Y 267.215,Z 463.051,A -85,B 0,C 180,E1 5571.501,E2 5571.501} C_VEL
LIN {X 0,Y 265.22,Z 460.039,A -85,B 0,C 180,E1 5568.475,E2 5568.475} C_VEL
LIN {X 0,Y 262.452,Z 456.389,A -85,B 0,C 180,E1 5561.557,E2 5561.557} C_VEL
LIN {X 0,Y 261.942,Z 456.612,A -85,B 0,C 180,E1 5558.505,E2 5558.505} C_VEL
LIN {X 0,Y 262.48,Z 459.83,A -85,B 0,C 180,E1 5551.814,E2 5551.814} C_VEL
LIN {X 0,Y 263.85,Z 463.786,A -85,B 0,C 180,E1 5547.832,E2 5547.832} C_VEL
LIN {X 0,Y 265.938,Z 469.12,A -85,B 0,C 180,E1 5544.003,E2 5544.003} C_VEL
LIN {X 0,Y 268.561,Z 475.889,A -85,B 0,C 180,E1 5540.416,E2 5540.416} C_VEL
LIN {X 0,Y 269.562,Z 478.766,A -85,B 0,C 180,E1 5539.211,E2 5539.211} C_VEL
LIN {X 0,Y 268.792,Z 488.689,A -85,B 0,C 180,E1 5538.708,E2 5538.708} C_VEL
LIN {X 0,Y 250.095,Z 643.499,A -85,B 0,C 180,E1 5535.851,E2 5535.851} C_VEL
LIN {X 0,Y 245.667,Z 665.949,A -85,B 0,C 180,E1 5535.242,E2 5535.242} C_VEL
LIN {X 0,Y 239.986,Z 686.799,A -85,B 0,C 180,E1 5534.425,E2 5534.425} C_VEL
LIN {X 0,Y 233.026,Z 706.891,A -85,B 0,C 180,E1 5533.358,E2 5533.358} C_VEL
LIN {X 0,Y 224.851,Z 726.224,A -85,B 0,C 180,E1 5532.011,E2 5532.011} C_VEL
LIN {X 0,Y 215.103,Z 745.537,A -85,B 0,C 180,E1 5530.252,E2 5530.252} C_VEL
LIN {X 0,Y 204.69,Z 763.18,A -85,B 0,C 180,E1 5528.148,E2 5528.148} C_VEL
LIN {X 0,Y 193.841,Z 779.221,A -85,B 0,C 180,E1 5525.656,E2 5525.656} C_VEL
LIN {X 0,Y 182.167,Z 794.447,A -85,B 0,C 180,E1 5522.544,E2 5522.544} C_VEL
LIN {X 0,Y 169.535,Z 809.052,A -85,B 0,C 180,E1 5518.511,E2 5518.511} C_VEL
LIN {X 0,Y 157.119,Z 821.934,A -85,B 0,C 180,E1 5513.603,E2 5513.603} C_VEL
LIN {X 0,Y 145.953,Z 832.538,A -85,B 0,C 180,E1 5507.959,E2 5507.959} C_VEL
LIN {X 0,Y 136.167,Z 841.308,A -85,B 0,C 180,E1 5501.439,E2 5501.439} C_VEL
LIN {X 0,Y 127.713,Z 848.747,A -85,B 0,C 180,E1 5493.595,E2 5493.595} C_VEL
LIN {X 0,Y 121.489,Z 854.503,A -85,B 0,C 180,E1 5484.743,E2 5484.743} C_VEL
LIN {X 0,Y 117.783,Z 858.606,A -85,B 0,C 180,E1 5475.251,E2 5475.251} C_VEL
LIN {X 0,Y 116.53,Z 861.103,A -85,B 0,C 180,E1 5465.432,E2 5465.432} C_VEL
LIN {X 0,Y 117.594,Z 862.171,A -85,B 0,C 180,E1 5455.56,E2 5455.56} C_VEL
LIN {X 0,Y 121.652,Z 861.722,A -85,B 0,C 180,E1 5445.03,E2 5445.03} C_VEL
LIN {X 0,Y 128.541,Z 859.639,A -85,B 0,C 180,E1 5435.687,E2 5435.687} C_VEL
LIN {X 0,Y 138.341,Z 855.803,A -85,B 0,C 180,E1 5427.265,E2 5427.265} C_VEL
LIN {X 0,Y 151.222,Z 849.781,A -85,B 0,C 180,E1 5419.705,E2 5419.705} C_VEL
LIN {X 0,Y 164.789,Z 842.39,A -85,B 0,C 180,E1 5413.898,E2 5413.898} C_VEL
LIN {X 0,Y 179.252,Z 833.419,A -85,B 0,C 180,E1 5409.167,E2 5409.167} C_VEL
LIN {X 0,Y 194.75,Z 822.455,A -85,B 0,C 180,E1 5405.162,E2 5405.162} C_VEL
LIN {X 0,Y 209.592,Z 810.516,A -85,B 0,C 180,E1 5402.056,E2 5402.056} C_VEL
LIN {X 0,Y 224.297,Z 797.014,A -85,B 0,C 180,E1 5399.488,E2 5399.488} C_VEL
LIN {X 0,Y 238.195,Z 782.297,A -85,B 0,C 180,E1 5397.415,E2 5397.415} C_VEL
LIN {X 0,Y 251.146,Z 766.522,A -85,B 0,C 180,E1 5395.736,E2 5395.736} C_VEL
LIN {X 0,Y 263.36,Z 749.374,A -85,B 0,C 180,E1 5394.334,E2 5394.334} C_VEL
LIN {X 0,Y 266.071,Z 745.122,A -85,B 0,C 180,E1 5394.036,E2 5394.036} C_VEL
LIN {X 0,Y 261.109,Z 753.213,A -85,B 0,C 180,E1 5393.77,E2 5393.77} C_VEL
LIN {X 0,Y 254.958,Z 762.224,A -85,B 0,C 180,E1 5393.85,E2 5393.85} C_VEL
LIN {X 0,Y 247.615,Z 771.831,A -85,B 0,C 180,E1 5394.341,E2 5394.341} C_VEL
LIN {X 0,Y 240.958,Z 779.693,A -85,B 0,C 180,E1 5395.061,E2 5395.061} C_VEL
LIN {X 0,Y 226.461,Z 795.027,A -85,B 0,C 180,E1 5396.962,E2 5396.962} C_VEL
LIN {X 0,Y 210.97,Z 809.264,A -85,B 0,C 180,E1 5399.365,E2 5399.365} C_VEL
LIN {X 0,Y 196.094,Z 821.224,A -85,B 0,C 180,E1 5402.126,E2 5402.126} C_VEL
LIN {X 0,Y 180.196,Z 832.371,A -85,B 0,C 180,E1 5405.731,E2 5405.731} C_VEL
LIN {X 0,Y 164.566,Z 841.83,A -85,B 0,C 180,E1 5410.201,E2 5410.201} C_VEL
LIN {X 0,Y 150.407,Z 849.282,A -85,B 0,C 180,E1 5415.457,E2 5415.457} C_VEL
LIN {X 0,Y 136.373,Z 855.666,A -85,B 0,C 180,E1 5422.524,E2 5422.524} C_VEL
LIN {X 0,Y 125.289,Z 859.929,A -85,B 0,C 180,E1 5430.482,E2 5430.482} C_VEL
LIN {X 0,Y 116.479,Z 862.632,A -85,B 0,C 180,E1 5440.193,E2 5440.193} C_VEL
LIN {X 0,Y 110.961,Z 863.539,A -85,B 0,C 180,E1 5450.901,E2 5450.901} C_VEL
LIN {X 0,Y 108.757,Z 862.863,A -85,B 0,C 180,E1 5461.447,E2 5461.447} C_VEL
LIN {X 0,Y 109.23,Z 860.714,A -85,B 0,C 180,E1 5472.424,E2 5472.424} C_VEL
LIN {X 0,Y 112.414,Z 857.103,A -85,B 0,C 180,E1 5482.852,E2 5482.852} C_VEL
LIN {X 0,Y 118.274,Z 851.928,A -85,B 0,C 180,E1 5492.428,E2 5492.428} C_VEL
LIN {X 0,Y 127.072,Z 844.608,A -85,B 0,C 180,E1 5501.349,E2 5501.349} C_VEL
LIN {X 0,Y 136.965,Z 836.259,A -85,B 0,C 180,E1 5508.299,E2 5508.299} C_VEL
LIN {X 0,Y 148.36,Z 826.112,A -85,B 0,C 180,E1 5514.278,E2 5514.278} C_VEL
LIN {X 0,Y 160.996,Z 813.88,A -85,B 0,C 180,E1 5519.386,E2 5519.386} C_VEL
LIN {X 0,Y 173.04,Z 800.982,A -85,B 0,C 180,E1 5523.297,E2 5523.297} C_VEL
LIN {X 0,Y 185.295,Z 786.289,A -85,B 0,C 180,E1 5526.606,E2 5526.606} C_VEL
LIN {X 0,Y 197.195,Z 770.085,A -85,B 0,C 180,E1 5529.334,E2 5529.334} C_VEL
LIN {X 0,Y 208.553,Z 752.232,A -85,B 0,C 180,E1 5531.593,E2 5531.593} C_VEL
LIN {X 0,Y 218.774,Z 733.452,A -85,B 0,C 180,E1 5533.394,E2 5533.394} C_VEL
LIN {X 0,Y 227.687,Z 714,A -85,B 0,C 180,E1 5534.817,E2 5534.817} C_VEL
LIN {X 0,Y 235.204,Z 694.094,A -85,B 0,C 180,E1 5535.927,E2 5535.927} C_VEL
LIN {X 0,Y 241.609,Z 672.756,A -85,B 0,C 180,E1 5536.81,E2 5536.81} C_VEL
LIN {X 0,Y 246.598,Z 650.338,A -85,B 0,C 180,E1 5537.462,E2 5537.462} C_VEL
LIN {X 0,Y 250.533,Z 622.98,A -85,B 0,C 180,E1 5538.008,E2 5538.008} C_VEL
LIN {X 0,Y 266.969,Z 487.153,A -85,B 0,C 180,E1 5540.439,E2 5540.439} C_VEL
LIN {X 0,Y 267.196,Z 483.989,A -85,B 0,C 180,E1 5540.635,E2 5540.635} C_VEL
LIN {X 0,Y 264.547,Z 476.812,A -85,B 0,C 180,E1 5544.407,E2 5544.407} C_VEL
LIN {X 0,Y 262.6,Z 471.541,A -85,B 0,C 180,E1 5548.175,E2 5548.175} C_VEL
LIN {X 0,Y 261.253,Z 467.221,A -85,B 0,C 180,E1 5552.551,E2 5552.551} C_VEL
LIN {X 0,Y 261.087,Z 464.226,A -85,B 0,C 180,E1 5559.84,E2 5559.84} C_VEL
LIN {X 0,Y 261.706,Z 464.796,A -85,B 0,C 180,E1 5562.777,E2 5562.777} C_VEL
LIN {X 0,Y 264.617,Z 468.731,A -85,B 0,C 180,E1 5569.247,E2 5569.247} C_VEL
LIN {X 0,Y 267.514,Z 473.238,A -85,B 0,C 180,E1 5573.24,E2 5573.24} C_VEL
LIN {X 0,Y 270.979,Z 478.781,A -85,B 0,C 180,E1 5576.934,E2 5576.934} C_VEL
LIN {X 0,Y 274.562,Z 485.074,A -85,B 0,C 180,E1 5580.131,E2 5580.131} C_VEL
LIN {X 0,Y 256.889,Z 651.217,A -85,B 0,C 180,E1 5583.209,E2 5583.209} C_VEL
LIN {X 0,Y 252.753,Z 673.305,A -85,B 0,C 180,E1 5583.744,E2 5583.744} C_VEL
LIN {X 0,Y 247.143,Z 694.458,A -85,B 0,C 180,E1 5584.375,E2 5584.375} C_VEL
LIN {X 0,Y 240.454,Z 714.432,A -85,B 0,C 180,E1 5585.176,E2 5585.176} C_VEL
LIN {X 0,Y 231.74,Z 735.55,A -85,B 0,C 180,E1 5586.302,E2 5586.302} C_VEL
LIN {X 0,Y 221.97,Z 755.177,A -85,B 0,C 180,E1 5587.684,E2 5587.684} C_VEL
LIN {X 0,Y 210.841,Z 774.374,A -85,B 0,C 180,E1 5589.452,E2 5589.452} C_VEL
LIN {X 0,Y 199.014,Z 792.11,A -85,B 0,C 180,E1 5591.594,E2 5591.594} C_VEL
LIN {X 0,Y 186.177,Z 809.063,A -85,B 0,C 180,E1 5594.304,E2 5594.304} C_VEL
LIN {X 0,Y 173.081,Z 824.372,A -85,B 0,C 180,E1 5597.593,E2 5597.593} C_VEL
LIN {X 0,Y 159.417,Z 838.898,A -85,B 0,C 180,E1 5601.828,E2 5601.828} C_VEL
LIN {X 0,Y 146.741,Z 851.313,A -85,B 0,C 180,E1 5606.79,E2 5606.79} C_VEL
LIN {X 0,Y 134.665,Z 862.384,A -85,B 0,C 180,E1 5612.959,E2 5612.959} C_VEL
LIN {X 0,Y 123.825,Z 872.145,A -85,B 0,C 180,E1 5620.615,E2 5620.615} C_VEL
LIN {X 0,Y 115.341,Z 880.163,A -85,B 0,C 180,E1 5629.441,E2 5629.441} C_VEL
LIN {X 0,Y 109.387,Z 886.709,A -85,B 0,C 180,E1 5639.813,E2 5639.813} C_VEL
LIN {X 0,Y 106.592,Z 891.73,A -85,B 0,C 180,E1 5651.396,E2 5651.396} C_VEL
LIN {X 0,Y 106.585,Z 894.422,A -85,B 0,C 180,E1 5660.818,E2 5660.818} C_VEL
LIN {X 0,Y 107.289,Z 895.56,A -85,B 0,C 180,E1 5667.858,E2 5667.858} C_VEL
LIN {X 0,Y 107.213,Z 895.743,A -85,B 0,C 180,E1 5672.667,E2 5672.667} C_VEL
LIN {X 0,Y 106.378,Z 895.164,A -85,B 0,C 180,E1 5680.281,E2 5680.281} C_VEL
LIN {X 0,Y 106.566,Z 893.265,A -85,B 0,C 180,E1 5690.307,E2 5690.307} C_VEL
LIN {X 0,Y 110.087,Z 889.299,A -85,B 0,C 180,E1 5702.396,E2 5702.396} C_VEL
LIN {X 0,Y 117.58,Z 883.722,A -85,B 0,C 180,E1 5713.527,E2 5713.527} C_VEL
LIN {X 0,Y 128.936,Z 876.148,A -85,B 0,C 180,E1 5723.335,E2 5723.335} C_VEL
LIN {X 0,Y 142.709,Z 867.158,A -85,B 0,C 180,E1 5731.128,E2 5731.128} C_VEL
LIN {X 0,Y 158.193,Z 856.664,A -85,B 0,C 180,E1 5737.327,E2 5737.327} C_VEL
LIN {X 0,Y 175.222,Z 844.182,A -85,B 0,C 180,E1 5742.34,E2 5742.34} C_VEL
LIN {X 0,Y 191.609,Z 830.894,A -85,B 0,C 180,E1 5746.055,E2 5746.055} C_VEL
LIN {X 0,Y 208.703,Z 815.515,A -85,B 0,C 180,E1 5749.129,E2 5749.129} C_VEL
LIN {X 0,Y 224.464,Z 799.579,A -85,B 0,C 180,E1 5751.426,E2 5751.426} C_VEL
LIN {X 0,Y 239.127,Z 782.752,A -85,B 0,C 180,E1 5753.217,E2 5753.217} C_VEL
LIN {X 0,Y 248.219,Z 771.092,A -85,B 0,C 180,E1 5754.208,E2 5754.208} C_VEL
LIN {X 0,Y 240.958,Z 779.693,A -85,B 0,C 180,E1 5755.061,E2 5755.061} C_VEL
LIN {X 0,Y 237.425,Z 783.807,A -85,B 0,C 180,E1 5755.274,E2 5755.274} C_VEL
LIN {X 0,Y 233.04,Z 788.782,A -85,B 0,C 180,E1 5755.09,E2 5755.09} C_VEL
LIN {X 0,Y 226.481,Z 795.992,A -85,B 0,C 180,E1 5754.228,E2 5754.228} C_VEL
LIN {X 0,Y 217.485,Z 805.371,A -85,B 0,C 180,E1 5752.785,E2 5752.785} C_VEL
LIN {X 0,Y 200.773,Z 821.022,A -85,B 0,C 180,E1 5750.397,E2 5750.397} C_VEL
LIN {X 0,Y 184.202,Z 834.885,A -85,B 0,C 180,E1 5747.459,E2 5747.459} C_VEL
LIN {X 0,Y 165.948,Z 848.437,A -85,B 0,C 180,E1 5743.32,E2 5743.32} C_VEL
LIN {X 0,Y 148.703,Z 859.99,A -85,B 0,C 180,E1 5738.096,E2 5738.096} C_VEL
LIN {X 0,Y 131.644,Z 870.563,A -85,B 0,C 180,E1 5730.851,E2 5730.851} C_VEL
LIN {X 0,Y 117.814,Z 878.831,A -85,B 0,C 180,E1 5722.108,E2 5722.108} C_VEL
LIN {X 0,Y 106.818,Z 885.584,A -85,B 0,C 180,E1 5710.929,E2 5710.929} C_VEL
LIN {X 0,Y 100.408,Z 890.278,A -85,B 0,C 180,E1 5698.547,E2 5698.547} C_VEL
LIN {X 0,Y 98.274,Z 893.279,A -85,B 0,C 180,E1 5685.938,E2 5685.938} C_VEL
LIN {X 0,Y 98.907,Z 894.386,A -85,B 0,C 180,E1 5675.796,E2 5675.796} C_VEL
LIN {X 0,Y 99.475,Z 894.487,A -85,B 0,C 180,E1 5669.994,E2 5669.994} C_VEL
LIN {X 0,Y 98.988,Z 893.819,A -85,B 0,C 180,E1 5664.197,E2 5664.197} C_VEL
LIN {X 0,Y 98.453,Z 891.789,A -85,B 0,C 180,E1 5654.684,E2 5654.684} C_VEL
LIN {X 0,Y 100.117,Z 887.808,A -85,B 0,C 180,E1 5643.288,E2 5643.288} C_VEL
LIN {X 0,Y 105.209,Z 881.998,A -85,B 0,C 180,E1 5631.843,E2 5631.843} C_VEL
LIN {X 0,Y 113.662,Z 874.374,A -85,B 0,C 180,E1 5621.599,E2 5621.599} C_VEL
LIN {X 0,Y 124.72,Z 864.976,A -85,B 0,C 180,E1 5613.036,E2 5613.036} C_VEL
LIN {X 0,Y 137.887,Z 853.636,A -85,B 0,C 180,E1 5605.943,E2 5605.943} C_VEL
LIN {X 0,Y 151.587,Z 841.108,A -85,B 0,C 180,E1 5600.499,E2 5600.499} C_VEL
LIN {X 0,Y 165.802,Z 826.871,A -85,B 0,C 180,E1 5596.106,E2 5596.106} C_VEL
LIN {X 0,Y 179.402,Z 811.7,A -85,B 0,C 180,E1 5592.743,E2 5592.743} C_VEL
LIN {X 0,Y 192.892,Z 794.759,A -85,B 0,C 180,E1 5589.967,E2 5589.967} C_VEL
LIN {X 0,Y 204.965,Z 777.594,A -85,B 0,C 180,E1 5587.851,E2 5587.851} C_VEL
LIN {X 0,Y 216.641,Z 758.502,A -85,B 0,C 180,E1 5586.068,E2 5586.068} C_VEL
LIN {X 0,Y 226.738,Z 739.07,A -85,B 0,C 180,E1 5584.7,E2 5584.7} C_VEL
LIN {X 0,Y 235.445,Z 719.234,A -85,B 0,C 180,E1 5583.625,E2 5583.625} C_VEL
LIN {X 0,Y 242.712,Z 699.245,A -85,B 0,C 180,E1 5582.796,E2 5582.796} C_VEL
LIN {X 0,Y 248.951,Z 677.351,A -85,B 0,C 180,E1 5582.139,E2 5582.139} C_VEL
LIN {X 0,Y 253.346,Z 655.76,A -85,B 0,C 180,E1 5581.628,E2 5581.628} C_VEL
LIN {X 0,Y 257,Z 626.369,A -85,B 0,C 180,E1 5581.049,E2 5581.049} C_VEL
LIN {X 0,Y 271.598,Z 490.31,A -85,B 0,C 180,E1 5578.577,E2 5578.577} C_VEL
LIN {X 0,Y 268.029,Z 484.04,A -85,B 0,C 180,E1 5575.079,E2 5575.079} C_VEL
